this function will calculate the trend of a given array.
trend will calculate the avg of the first half of the array and then the avg of the second half, trend = avg2 - avg1.
for example:  [0,1,4,5,3,4,6,3] = 4 - 2.5 = 1.5
the function needs to be called:	array_trend(adr("array"),sizeof("array"));
because this function works with pointers its very time efficient and it needs no extra memory.

*)
stop := SHR(size,2)-1;
stop2 := SHR(stop,1);
FOR i := 0 TO stop2 DO x := x - pt^[i]; END_FOR;
IF EVEN(UINT_TO_INT(stop)) THEN
	FOR i := stop2 TO stop DO X := X + pt^[i]; END_FOR;
ELSE
	FOR i := stop2 + 1 TO stop DO X := X + pt^[i]; END_FOR;
END_IF;
ARRAY_TREND := x / (stop2 + 1);

(* revision history
hm	2 oct 2007	rev 1.0
	original version

hm	12 dec 2007	rev 1.1
	changed code for better performance

hm	16. mar. 2008	rev 1.2
	changed type of input size to uint

*)
END_FUNCTION

(* POU ASINH, ST *)
FUNCTION ASINH : REAL
VAR_INPUT
	X : REAL;
END_VAR
VAR
END_VAR


(*
version 1.2	16. mar 2008
programmer 	hugo
tested by		tobias

this function calculates the arcus sin hyperbolicus

*)
ASINH := LN(SQRT(X * X + 1)+X);

(* revision history
hm		12 jan 2007	rev 1.0
	original version

hm		2. dec 2007	rev 1.1
	changed code for better performance

hm		16.3. 2007		rev 1.2
	changed sequence of calculations to improve performance

*)
END_FUNCTION

(* POU ASTRO, ST *)
FUNCTION_BLOCK ASTRO
VAR_INPUT
	m : REAL;
	AE : REAL;
	PC : REAL;
	LJ : REAL;
END_VAR
VAR_OUTPUT
	Ym : REAL;
	YAE : REAL;
	YPC : REAL;
	YLJ : REAL;
END_VAR
VAR
END_VAR

(*
version 1.0	27 mar 2007
programmer 	hugo
tested by		oscat

this function converts different length units
any unused input can simply be left open.
different inputs connected at the same time will be added up.

*)
YAE :=	AE
		+ m / 149.597870E9
		+ PC * 206265
		+ LJ * 63240;
Ym := YAE * 149.597870E9;
YPC := YAE / 206265;
YLJ := YAE / 63240;


(*
Länge Meter m SI-Basiseinheit
Astronomische Einheit* AE 1 AE = 149,597 870 · E9 m
Parsec pc 1 pc = 206265 AE = 30,857 · E15 m
Lichtjahr Lj 1 Lj = 9,460 530 · E15 m = 63240 AE = 0,306 59 pc
Ångström Å 1 Å = E–l0 m
typograph. Punkt p 1 p = 0,376 065 mm • im Druckereigewerbe
inch** in 1 in = 2,54 · E–2 m = 25,4 mm***
foot ft 1 ft = 0,3048 m = 30,48 cm
yard yd 1 yd = 0,9144 m
mile mile 1 mile = 1609,344 m
Internat. Seemeile sm 1 sm = 1852 m
Fathom fm 1 fm = 1,829 m • in der Seeschifffahrt

*)
END_FUNCTION_BLOCK

(* POU ATAN2, ST *)
FUNCTION ATAN2 : REAL
VAR_INPUT
	Y : REAL;
	X : REAL;
END_VAR
VAR
END_VAR


(*
version 1.1	18. oct. 2008
programmer 	hugo
tested by	oscat

this function calculates the angle in a coordinate system in rad.

*)
IF X > 0 THEN
	ATAN2 := ATAN(Y/X);
ELSIF X < 0 THEN
	IF Y >=0 THEN
		ATAN2 := ATAN(Y/X) + MATH.PI;
	ELSE
		ATAN2 := ATAN(Y/X) - MATH.PI;
	END_IF;
ELSIF Y > 0 THEN
	ATAN2 := MATH.PI05;
ELSIF Y < 0 THEN
	ATAN2 := -MATH.PI05;
ELSE
	ATAN2 := 0;
END_IF;


(* revision history
hm	20.  apr. 2008	rev 1.0
	original version

hm	18. oct. 2008	rev 1.1
	changed to use math constants
*)
END_FUNCTION

(* POU ATANH, ST *)
FUNCTION ATANH : REAL
VAR_INPUT
	X : REAL;
END_VAR
VAR
END_VAR


(*
version 1.1	5. jan 2008
programmer 	hugo
tested by		tobias

this function calculates the arcus tangens hyperbolicus

*)
ATANH := LN((1+x)/(1-x)) * 0.5;


(* revision history
hm		12 jan 2007	rev 1.0
	original version

hm		5. jan 2008	rev 1.1
	improved code for better performance
*)
END_FUNCTION

(* POU B_TRIG, ST *)
FUNCTION_BLOCK B_TRIG
VAR_INPUT
	CLK : BOOL;
END_VAR
VAR_OUTPUT
	Q : BOOL;
END_VAR
VAR
	edge : BOOL;
END_VAR

(*
version 1.0	4. aug. 2006
programmer 	hugo
tested by		tobias

this block is similar to R_trig and F_trig but it generates a pulse on rising and falling edge.

*)
Q := clk XOR edge;
edge := CLK;


(* revision history
hm		4. aug. 2006	rev 1.0
	original version

*)
END_FUNCTION_BLOCK

(* POU BAR_GRAPH, ST *)
FUNCTION_BLOCK BAR_GRAPH
VAR_INPUT
	X : REAL;
	rst : BOOL;
END_VAR
VAR_INPUT CONSTANT
	trigger_Low : REAL;
	trigger_High : REAL;
	Alarm_low : BOOL;
	Alarm_high : BOOL;
	log_scale : BOOL;
END_VAR
VAR_OUTPUT
	LOW, Q1, Q2, Q3, Q4, Q5, Q6, HIGH : BOOL;
	Alarm : BOOL;
	Status : BYTE;
END_VAR
VAR
	init : BOOL;
	T1, T2, T3, T4, T5 : REAL;
END_VAR
VAR_TEMP
	temp : REAL;
END_VAR

(*
	version 1.2	6 jan 2008
	programmer 	hugo
	tested BY		hans

bar graph is a muti window comparator which displays an analog input signal on 8 digital outputs.
only one output is active a any given time depending on the value of the input signal.
the output can be of linear or logarithmic scale.

*)
IF NOT init THEN
	init := TRUE;
	IF log_scale THEN
		temp := EXP(LN(Trigger_high / Trigger_low) * 0.166666666666666666666);
		T1 := trigger_low * temp;
		T2 := T1 * temp;
		T3 := T2 * temp;
		T4 := T3 * temp;
		T5 := T4 * temp;
	ELSE
		temp := (trigger_high - trigger_low) * 0.142857142;
		T1 := trigger_low + temp;
		T2 := T1 + temp;
		T3 := T2 + temp;
		T4 := T3 + temp;
		T5 := T4 + temp;
	END_IF;
END_IF;

(* clear outputs before checking *)
Q1 := FALSE;
Q2 := FALSE;
Q3 := FALSE;
Q4 := FALSE;
Q5 := FALSE;
Q6 := FALSE;
status := 110;

(* low, high and alarm can only be cleared with rst depending on alarm_low and alarm_high *)
IF NOT alarm_low THEN low := FALSE; END_IF;
IF NOT alarm_high THEN high := FALSE; END_IF;
IF rst THEN
	alarm := FALSE;
	low := FALSE;
	high := FALSE;
END_IF;

(* check and set outputs *)
IF X < trigger_low THEN
	Low := TRUE;
	status := 111;
	IF alarm_low THEN
		alarm := TRUE;
		status := 1;
	END_IF;
ELSIF X < T1 THEN
	Q1 := TRUE;
ELSIF x < t2 THEN
	Q2 := TRUE;
ELSIF x < t3 THEN
	Q3 := TRUE;
ELSIF x < T4 THEN
	Q4 := TRUE;
ELSIF x < T5 THEN
	q5 := TRUE;
ELSIF x < trigger_high THEN
	q6 := TRUE;
ELSE
	high := TRUE;
	status := 112;
	IF alarm_high THEN
		alarm := TRUE;
		status := 2;
	END_IF;
END_IF;

(* revision history
hm	22. feb 2007	rev 1.0
	original version

hm	2. dec 2007		rev 1.1
	chaged code for better performance

hm	6. jan 2008		rev 1.2
	further performance improvement

*)
END_FUNCTION_BLOCK

(* POU BCDC_TO_INT, ST *)
FUNCTION BCDC_TO_INT : INT
VAR_INPUT
	IN : BYTE;
END_VAR
VAR
END_VAR

(*
version 1.1 30. jun. 2008
programmer 	hugo
tested by	oscat

this function converts a two digit bcd number into an integer.

*)
BCDC_TO_INT := (in AND 16#0F) + (SHR(in,4) * 10);

(* revision history
hm	13.12.2007	rev 1.0
	original version

hm	30.6.2008	rev 1.1
	changed name BCD_TO_INT to BCDC_TO_INT to avoid collision with util.lib

*)
END_FUNCTION

(* POU BETA, ST *)
FUNCTION BETA : REAL
VAR_INPUT
	X : REAL;
	Y : REAL;
END_VAR
VAR
END_VAR

(*
version 1.0	26. oct. 2008
programmer 	hugo
tested by		oscat

this function calculates the beta function for real number > 0.

*)
BETA := GAMMA(X) * GAMMA(Y) / GAMMA(x + y);


(* revision history
hm	26. oct. 2008	rev 1.0
	original version

*)
END_FUNCTION

(* POU GAMMA, ST *)
FUNCTION GAMMA : REAL
VAR_INPUT
	X : REAL;
END_VAR
VAR
END_VAR

(*
version 1.2	26. oct. 2008
programmer 	hugo
tested by	oscat

this function calculates the stirling function which is an approximation for the gamma function

*)
IF x > 0 THEN
	GAMMA := SQRT(math.PI2/X) * EXPT(math.E_INV * (x + 1 / (12 * x - 0.1 / X)),x);
END_IF;


(* the stirling formula is not very accurate for small values of X
IF X >=0 THEN GAMMA := SQRT(math.PI2 * X) * EXPT(X / math.E, X); END_IF;
*)





(* revision history
hm	10.12.2007	rev 1.0
	original version

hm	18. oct. 2008	rev 1.1
	using math constants

hm	26. oct. 2008	rev 1.2
	using new formula with better accuracy
*)
END_FUNCTION

(* POU BFT_TO_MS, ST *)
FUNCTION BFT_TO_MS : REAL
VAR_INPUT
	BFT : INT;
END_VAR
VAR
END_VAR

(*
version 1.0	12. jun 2008
programmer 	hugo
tested by	oscdat

this function converts wind speed from beaufort to m/s
*)
BFT_TO_MS := EXPT(BFT, 1.5) * 0.836;


(* revision history
hm	12. 6. 2008		rev 1.0
	original version

*)
END_FUNCTION

(* POU BIN_TO_BYTE, ST *)
FUNCTION BIN_TO_BYTE : BYTE
VAR_INPUT
	BIN : STRING(12);
END_VAR
VAR
	pt : POINTER TO BYTE;
	i: INT;
	X: BYTE;
	stop: INT;
END_VAR

(*
version 1.1	20. sep. 2008
programmer 	hugo
tested by	oscat

BINARY_TO_byte converts a binary string into a byte.

*)
pt := ADR(bin);
stop := LEN(bin);
FOR I := 1 TO stop DO
	(* read the first character and subtract 48 to get value in decimal 0 = 48 *)
	x := pt^;
	(* calculate the value of the digit *)
	IF X = 48 OR X = 49 THEN
		BIN_TO_BYTE := SHL(BIN_TO_BYTE,1) + X - 48;
	END_IF;
	pt := pt + 1;
END_FOR;



(* revision histroy
hm	18. jun. 2008	rev 1.0
	original release

hm	20. sep. 2008	rev 1.1
	changed length of input string from 20 to 12

*)	
END_FUNCTION

(* POU BIN_TO_DWORD, ST *)
FUNCTION BIN_TO_DWORD : DWORD
VAR_INPUT
	BIN : STRING(40);
END_VAR
VAR
	pt : POINTER TO BYTE;
	i: INT;
	X: BYTE;
	stop: INT;
END_VAR

(*
version 1.1	20. sep. 2008
programmer 	hugo
tested by	oscat

BINARY_TO_DWORD converts a binary string into a dword.

*)
pt := ADR(bin);
stop := LEN(bin);
FOR I := 1 TO stop DO
	(* read the first character and subtract 48 to get value in decimal 0 = 48 *)
	x := pt^;
	(* calculate the value of the digit *)
	IF X = 48 OR X = 49 THEN
		BIN_TO_DWORD := SHL(BIN_TO_DWORD,1) + X - 48;
	END_IF;
	pt := pt + 1;
END_FOR;



(* revision histroy
hm	18. jun. 2008	rev 1.0
	original release

hm	20. sep. 2008	rev 1.1
	changed length of input dtring from 20 to 40
*)	
END_FUNCTION

(* POU BINOM, ST *)
FUNCTION BINOM : DINT
VAR_INPUT
	N : INT;
	K : INT;
END_VAR

VAR
	i: INT;
END_VAR


(*
version 1.0	25. oct. 2008
programmer 	hugo
tested by		tobias

this function calculates the binomialkoefficient (N over k)

*)
IF 2 * K > n THEN
	k := n - k;
END_IF;
IF k > n THEN
	RETURN;
ELSIF k = 0 OR k = n THEN
	BINOM := 1;
ELSIF k = 1 THEN
	BINOM := n;
ELSE
	BINOM := n;
	n := n + 1;
	FOR i := 2 TO k DO
		BINOM := BINOM * (n - i) / i;
	END_FOR
END_IF;



(*
binomialkoeffizient(n, k)
1  wenn k = 0 return 1
2  wenn 2k > n
3      dann führe aus ergebnis \leftarrow binomialkoeffizient(n, n-k)
4  sonst führe aus ergebnis \leftarrow n
5          von i \leftarrow 2 bis k
6              führe aus ergebnis \leftarrow ergebnis \cdot (n + 1 - i)
7                        ergebnis \leftarrow ergebnis : i
8  return ergebnis
*)



(* revision history
hm	25. oct. 2008	rev 1.0
	original version


*)
END_FUNCTION

(* POU BIT_LOAD_B, ST *)
FUNCTION BIT_LOAD_B : BYTE
VAR_INPUT
	IN : BYTE;
	VAL : BOOL;
	POS : INT;
END_VAR
VAR CONSTANT
	dat : BYTE := 1;
END_VAR

(*
version 1.1	16. mar 2008
programmer 	hugo
tested by	tobias

this function loads a bit into a byte at position pos.
 *)
IF VAL THEN
	BIT_LOAD_B := in OR SHL(dat,pos);
ELSE
	BIT_LOAD_B := in AND (NOT SHL(dat,pos));
END_IF;


(* revision history
hm	29. feb 2008	rev 1.0
	original version

hm	16. mar 2008	rev 1.1
	change input bit to val for compatibility reasons
*)
END_FUNCTION

(* POU BIT_LOAD_B2, ST *)
FUNCTION BIT_LOAD_B2 : BYTE
VAR_INPUT
	I : BYTE;
	D : BOOL;
	P : INT;
	N : INT;
END_VAR


(*
version 1.0 18. oct. 2008
programmer 	hugo
tested by	tobias

this function loads N bits of D at pos P in Byte I

*)
IF D THEN
	BIT_LOAD_B2 := ROL(SHR(BYTE#255, 8 - N) OR ROR(i, P), P);
ELSE
	BIT_LOAD_B2 := ROL(SHL(BYTE#255, N) AND ROR(I, P), P);
END_IF;



(* revision history
hm	18. oct. 2008	rev 1.0
	original version


*)
END_FUNCTION

(* POU BIT_LOAD_DW, ST *)
FUNCTION BIT_LOAD_DW : DWORD
VAR_INPUT
	IN : DWORD;
	VAL : BOOL;
	POS : INT;
END_VAR
VAR CONSTANT
	dat : DWORD := 1;
END_VAR

(*
version 1.1	16. mar 2008
programmer 	hugo
tested by	tobias

this function loads a bit into a DWord at position pos.
 *)
IF val THEN
	BIT_LOAD_DW := in OR SHL(dat,pos);
ELSE
	BIT_LOAD_DW := in AND (NOT SHL(dat,pos));
END_IF;


(* revision history
hm	29. feb 2008	rev 1.0
	original version

hm	16. mar 2008	rev 1.1
	change input bit to val for compatibility reasons
*)
END_FUNCTION

(* POU BIT_LOAD_DW2, ST *)
FUNCTION BIT_LOAD_DW2 : DWORD
VAR_INPUT
	I : DWORD;
	D : BOOL;
	P : INT;
	N : INT;
END_VAR


(*
version 1.0 18. oct. 2008
programmer 	hugo
tested by	tobias

this function loads N bits of D at pos P in DWORD I

*)
IF D THEN
	BIT_LOAD_DW2 := ROL(SHR(DWORD#4294967295, 32 - N) OR ROR(i, P), P);
ELSE
	BIT_LOAD_DW2 := ROL(SHL(DWORD#4294967295, N) AND ROR(I, P), P);
END_IF;



(* revision history
hm	18. oct. 2008	rev 1.0
	original version


*)
END_FUNCTION

(* POU BIT_LOAD_W, ST *)
FUNCTION BIT_LOAD_W : WORD
VAR_INPUT
	IN : WORD;
	VAL : BOOL;
	POS : INT;
END_VAR
VAR CONSTANT
	dat : WORD := 1;
END_VAR

(*
version 1.1	16. mar 2008
programmer 	hugo
tested by	tobias

this function loads a bit into a Word at position pos.
 *)
IF val THEN
	BIT_LOAD_W := in OR SHL(dat,pos);
ELSE
	BIT_LOAD_W := in AND (NOT SHL(dat,pos));
END_IF;


(* revision history
hm	29. feb 2008	rev 1.0
	original version

hm	16. mar 2008	rev 1.1
	change input bit to val for compatibility reasons
*)
END_FUNCTION

(* POU BIT_LOAD_W2, ST *)
FUNCTION BIT_LOAD_W2 : WORD
VAR_INPUT
	I : WORD;
	D : BOOL;
	P : INT;
	N : INT;
END_VAR


(*
version 1.0 18. oct. 2008
programmer 	hugo
tested by	tobias

this function loads N bits of D at pos P in WORD I

*)
IF D THEN
	BIT_LOAD_W2 := ROL(SHR(WORD#65535, 16 - N) OR ROR(i, P), P);
ELSE
	BIT_LOAD_W2 := ROL(SHL(WORD#65535, N) AND ROR(I, P), P);
END_IF;



(* revision history
hm	18. oct. 2008	rev 1.0
	original version


*)
END_FUNCTION

(* POU BIT_OF_DWORD, ST *)
FUNCTION BIT_OF_DWORD : BOOL
VAR_INPUT
	in : DWORD;
	N : INT;
END_VAR
VAR
END_VAR

(*
version 1.2	6. jun. 2008
programmer 	hugo
tested by	tobias

this function extracts a single bit from the nth position from right (right is lowest bit)
the lowest Bit (Bit0 from in) is selected with N=0.
 *)
BIT_OF_DWORD := (SHR(in,N) AND 16#00000001) > 0;


(* old code used before rev 1.1
temp := SHR(in,n);
Bit_of_Dword := temp.0;
*)


(* revision history
hm	4. aug. 2006	rev 1.0
	original version

hm	29. feb 2008	rev 1.1
	improved performance

hm	6. jun. 2008	rev 1.2
	changes type of input N from byte to int
*)
END_FUNCTION

(* POU BIT_TOGGLE_B, ST *)
FUNCTION BIT_TOGGLE_B : BYTE
VAR_INPUT
	IN : BYTE;
	POS : INT;
END_VAR


(*
version 1.0 18. oct. 2008
programmer 	hugo
tested by	tobias

this function toggles a bit of a BYTE at position pos.

*)
BIT_TOGGLE_B := SHL(BYTE#1, POS) XOR IN;




(* revision history
hm	18. oct. 2008	rev 1.0
	original version


*)
END_FUNCTION

(* POU BIT_TOGGLE_DW, ST *)
FUNCTION BIT_TOGGLE_DW : DWORD
VAR_INPUT
	IN : DWORD;
	POS : INT;
END_VAR


(*
version 1.0 18. oct. 2008
programmer 	hugo
tested by	tobias

this function toggles a bit of a WORD at position pos.

*)
BIT_TOGGLE_DW := SHL(DWORD#1, POS) XOR IN;



(* revision history
hm	18. oct. 2008	rev 1.0
	original version


*)
END_FUNCTION

(* POU BIT_TOGGLE_W, ST *)
FUNCTION BIT_TOGGLE_W : WORD
VAR_INPUT
	IN : WORD;
	POS : INT;
END_VAR


(*
version 1.0 18. oct. 2008
programmer 	hugo
tested by	tobias

this function toggles a bit of a WORD at position pos.

*)
BIT_TOGGLE_W := SHL(WORD#1, POS) XOR IN;



(* revision history
hm	18. oct. 2008	rev 1.0
	original version


*)
END_FUNCTION

(* POU BLIND_ACTUATOR, ST *)
 FUNCTION_BLOCK BLIND_ACTUATOR
VAR_INPUT
	UP, DN : BOOL;
	S_IN : BYTE;
	T_UD : TIME := T#10s;
	T_ANGLE : TIME := T#3s;
END_VAR
VAR_INPUT CONSTANT
	T_LOCKOUT : TIME := t#100ms;
END_VAR
VAR_OUTPUT
	POS, ANG : BYTE;
	QU, QD : BOOL;
	STATUS : BYTE;
END_VAR
VAR
	position, angle : RMP_B;
	lock : INTERLOCK;
END_VAR

(*
version 1.2	18. oct. 2008
programmer 	hugo
tested by	oscat

blind actuator drives the up and down motor of a blind. T_lockout specifies the time between up or dn becomes active. 
To change direction there must be a minimum wait time to allow the motors to come to rest first.
the up and down outputs QU and QD are controlled by the inputs UP and DN.
the outputs pos and ang simulate the position of the blind pos = 0 means blind is down and pos = 255 = blind is up.
the angle 0 means vertical posisition of the slates and 255 means horizontal position of the slates.


*)
(* make sure only one motor is active at a given time *)
lock(i1 := UP, I2 := DN, TL := T_lockout);

(* ramp up or down to simulate the angle position of the blind slats *)
angle(e := lock.Q1 OR lock.Q2, UP := lock.Q1, PT := T_Angle);
position(e := lock.Q1 AND angle.high OR lock.Q2 AND angle.low, up := lock.Q1, PT := T_UD);

(* set the outputs *)
pos := position.Out;
ang := angle.Out;
QU := lock.Q1;
QD := lock.Q2;

(* set the status output *)
IF UP AND DN THEN
	IF s_in < 10 AND S_in > 1 THEN status := s_in; ELSE status := 1; END_IF;			(* error up and down together are not allowed *)
ELSIF S_IN > 0 THEN
	status := S_IN;
ELSIF UP THEN
	status := 101;
ELSIF DN THEN
	status := 102;
ELSE
	status := 0;
END_IF;


(* revision history
hm	29. sep 2007	rev 1.0
	original release

hm	6. oct 2007		rev 1.1
	rearanged outputs

hm	18. oct. 2008	rev 1.2
	changed calls for rmp_B because of change in RMP_B
*)
END_FUNCTION_BLOCK

(* POU RMP_B, ST *)
FUNCTION_BLOCK RMP_B
VAR_INPUT
	SET : BOOL;
	PT : TIME;
	E : BOOL := TRUE;
	UP : BOOL := TRUE;
	RST : BOOL;
END_VAR
VAR_OUTPUT
	OUT : BYTE;
	BUSY: BOOL;
	HIGH : BOOL;
	LOW : BOOL;
END_VAR
VAR
	rmp : _RMP_B;
END_VAR


(*
version 2.0	23. oct. 2008
programmer 	oscat
tested BY	oscat

this ramp generator generates a byte wide ramp with 255 steps
the generator has an asynchronous set and reset
the ramp is controlled by PT which is the total ramp time for a full sweep from 0..255
an UD input controlls the direction Up or Down and the E input enables the ramp generation
a busy output indicates that the ramp is running, busy false means output is stable.
the outputs low and high will be true when the output has reached its max or min value.

*)
(* generate ramp *)
rmp(dir := UP, E := E, TR := PT, rmp := out);

(* set or reset operation *)
IF RST THEN
	out := 0;
ELSIF SET THEN
	out := 255;
END_IF;

(* checks for outputs stable and reset or set busy flag *)
low := out = 0;
high := out = 255;
busy := NOT (low OR high) AND E;


(* revision history

hm 5.10.2006	rev 1.1
	added busy output
hm 17.1.2007	rev 1.2
	renamed input ud to up for better usability
	deleted unused variable step

hm	17.9.2007		rev 1.3
	replaced time() with t_plc_ms() for compatibility reasons

hm	28. sep 2007	rev 1.4
	added outputs on and off
	busy is now disabled while en is false
	new coding for higher accuracy and performance

hm	5. oct 2007	rev 1.5
	added statements to allow for PT to be t#0s output jumps to max or min immediately

hm	25. dec 2007	rev 1.6
	improved code for better performance

hm	16. oct. 2008	rev 1.7
	improved code for better performance

hm	18. oct. 2008	rev 1.8
	added type conversion to avoid warnings
	changed input en to e for compatibility reasons

hm	23. oct. 2008	REV 	2.0
	new code using _RMP_B

*)
END_FUNCTION_BLOCK

(* POU INTERLOCK, ST *)
FUNCTION_BLOCK INTERLOCK
VAR_INPUT
	I1, I2 : BOOL;
	TL : TIME;
END_VAR
VAR_OUTPUT
	Q1, Q2 : BOOL;
END_VAR
VAR
	T1, T2 : TOF;
END_VAR

(*
version 1.0	28 sep 2007
programmer 	hugo
tested by		tobias

INTERLOCK has two inputs I1 and I2 which drive the corresponding outputs Q1 and Q2.
the inputs signals lock each other out and therfore I1 can only drive Q1 when I2 is Low and vice versa.
The input TL specifies a dead time between two outputs can become active.
an output can only become active when the other output was not active for the time TL.

*)
(* the input signal have a run delay to lockout the other input *)
T1(IN := I1, PT := TL);
T2(IN := I2, PT := TL);

Q1 := I1 AND NOT t2.Q;
Q2 := I2 AND NOT t1.Q;


(* revision history

hm	28 sep 2007		rev 1.0
	original version

*)
END_FUNCTION_BLOCK

(* POU BLIND_CONTROL, ST *)
FUNCTION_BLOCK BLIND_CONTROL
VAR_INPUT
	UP, DN : BOOL;
	S_IN : BYTE;
	PI : BYTE;
	AI : BYTE;
	T_UD, T_ANGLE : TIME;
END_VAR
VAR_INPUT CONSTANT
	SENS : BYTE := 5;
	T_LOCKOUT: TIME := T#100ms;
END_VAR
VAR_OUTPUT
	POS, ANG : BYTE;
	MU, MD : BOOL;
	STATUS : BYTE;
END_VAR
VAR
	act : BLIND_ACTUATOR;
	delta : BYTE;
END_VAR

(*
version 1.3	30. oct 2007
programmer 	hugo
tested by		tobias


*)
IF UP AND DN THEN
	(* automatic modus detected *)
	(* first find correct position *)
	IF BYTE_TO_INT(act.pos) < BYTE_TO_INT(pi) - delta THEN
		act.UP := TRUE;
		act.DN := FALSE;
		delta := 0;
		act.S_IN := 121;
	ELSIF BYTE_TO_INT(act.pos) > BYTE_TO_INT(pi) + delta THEN
		act.UP := FALSE;
		act.DN := TRUE;
		delta := 0;
		act.S_IN := 122;
	(* regulate angle *)
	ELSIF BYTE_TO_INT(act.ang) < BYTE_TO_INT(ai) - delta AND T_angle > T#100ms THEN
		act.UP := TRUE;
		act.DN := FALSE;
		delta := 0;
		act.S_IN := 123;
	ELSIF BYTE_TO_INT(act.ang) > BYTE_TO_INT(ai) + delta AND T_angle > T#100ms THEN
		act.UP := FALSE;
		act.DN := TRUE;
		delta := 0;
		act.S_IN := 124;
	(* correct position reached *)
	ELSE
		act.UP := FALSE;
		act.DN := FALSE;
		delta := sens;
		act.S_IN := 0;
	END_IF;
ELSE
	act.UP := UP;
	act.DN := DN;
END_IF;

(* hand over status *)
IF s_in > 0 THEN act.S_IN := S_IN; END_IF;

(* blind control calls blind_actuator *)
act(T_UD:=T_UD, T_ANGLE:=T_ANGLE, T_lockout := T_Lockout);
pos := act.pos;
ang := act.ang;
MU := act.QU;
md := act.QD;
status := act.status;

(* revision history
hm	29. sep 2007	rev 1.0
	original release

hm	6. oct 2007		rev 1.1
	rearranged outputs
	integrated blind_actuator into blind_control

hm	16. oct 2007	rev 1.2
	ignore angle when t_angle = 0

hm 29. oct 2007	rev 1.3
	added lockout configuration time for motor direction change
	sens has a setup value of 5
*)
END_FUNCTION_BLOCK

(* POU BLIND_INPUT, ST *)
FUNCTION_BLOCK BLIND_INPUT
VAR_INPUT
	POS, ANG : BYTE;
	S1, S2 : BOOL;
	IN : BOOL;
	PI, AI : BYTE;
END_VAR
VAR_INPUT CONSTANT
	SINGLE_SWITCH : BOOL;
	CLICK_EN : BOOL := TRUE;
	CLICK_TIME : TIME := T#500ms;
	MAX_RUNTIME : TIME := T#60s;
	MANUAL_TIMEOUT: TIME := T#1h;
	DEBOUNCE_TIME : TIME := T#20ms;
	DBL_CLK1 : BOOL := FALSE;
	DBL_POS1 : BYTE;
	DBL_ANG1 : BYTE;
	DBL_CLK2 : BOOL := FALSE;
	DBL_POS2 : BYTE := 255;
	DBL_ANG2 : BYTE := 255;
	D1_TOGGLE : BOOL := TRUE;
	D2_TOGGLE : BOOL := TRUE;
END_VAR
VAR_OUTPUT
	QU, QD : BOOL;
	STATUS : BYTE;
	PO, AO : BYTE;
	D1, D2 : BOOL;
END_VAR
VAR
	s1e, s2e : TOF;
	s1d, s2d : CLICK_MODE;
	dir : BOOL;
	tx, last : TIME;
END_VAR

(*
version 1.5	22. jan. 2009
programmer 	hugo
tested by		oscat


*)
(* read system timer *)
tx := DWORD_TO_TIME(T_PLC_MS());

(* inputs S1 and S2 are debounced and then decoded for multiple clicks *)
s1e(in := S1, pt := DEBOUNCE_TIME);
s2e(in := S2, pt := DEBOUNCE_TIME);
s1d(in := (s1e.Q AND NOT SINGLE_SWITCH) OR (s1e.Q AND SINGLE_SWITCH AND dir), t_long := CLICK_TIME);
s2d(in := (s2e.Q AND NOT SINGLE_SWITCH) OR (s1e.Q AND SINGLE_SWITCH AND NOT dir), t_long := CLICK_TIME);

(* if d1 and d2 are not toggle clear them to make sure they are only active for oine cycle *)
IF NOT d1_toggle THEN d1 := FALSE; END_IF;
IF NOT d2_toggle THEN d2 := FALSE; END_IF;

(* decode actions *)
IF s1d.tp_LONG THEN
	status := 132;
ELSIF s2d.tp_LONG THEN
	status := 133;
ELSIF  s1d.SINGLE THEN
	IF click_en THEN
		(* if running then we stop otherwise start new direction *)
		IF QU XOR QD THEN
			status := 131;
		ELSE
			status := 134;
			last := tx;
			dir := NOT dir;
		END_IF;
	END_IF;
ELSIF  s2d.SINGLE THEN
	IF click_en THEN
		(* if running then we stop otherwise start new direction *)
		IF QU XOR QD THEN
			status := 131;
		ELSE
			status := 135;
			last := tx;
			dir := NOT dir;
		END_IF;
	END_IF;
ELSIF in THEN
	status := 136;
	last := tx;
ELSIF s1d.DOUBLE THEN
	IF dbl_clk1 THEN
		(* a position need to be set for a double click on S1 *)
		status := 137;
		last := tx;
	ELSE
		(* toggle the output when dbl_clk1 is not active *)
		D1 := NOT D1;
	END_IF;
ELSIF s2d.DOUBLE THEN
	IF dbl_clk2 THEN
		(* a position need to be set for a double click on S2 *)
		status := 138;
		last := tx;
	ELSE
		(* toggle the output when dbl_clk2 is not active *)
		(* in single switch mode we need to toggle d1 instead of d2 *)
		IF single_switch THEN D1 := NOT D1; ELSE D2 := NOT D2; END_IF;
	END_IF;
END_IF;


(* state machine *)
CASE status OF
	0:	(* automatic standby operation *)
			QU := QD := TRUE;
			PO := POS; AO := ANG;
	131:	(* manual operation standby *)
			QU := QD := FALSE;
			(* manual mode will be ended when timeout is reached *)
			IF tx - last >= manual_timeout THEN status := 0; END_IF;
	132:	(* manual operation up *)
			QU := TRUE; QD := FALSE;
			PO := POS; AO := ANG;
			last := tx;
			IF NOT s1d.LONG THEN status := 131; dir := NOT dir; END_IF;
	133:	(* manual operation down *)
			QU := FALSE; QD := TRUE;
			PO := POS; AO := ANG;
			last := tx;
			IF NOT s2d.LONG THEN	status := 131; dir := NOT dir; END_IF;
	134:	(* manual operation single click up *)
			QU := TRUE; QD := FALSE;
			PO := POS; AO := ANG;
			IF tx - last >= max_runtime THEN status := 131; END_IF;
	135:	(* manual operation single click dn *)
			QU := FALSE; QD := TRUE;
			PO := POS; AO := ANG;
			IF tx - last >= max_runtime THEN status := 131;	END_IF;
	136:	(* forced input in = true *)
			QU := QD := TRUE;
			PO := PI; AO := AI;
			IF tx-last >= max_runtime THEN status := 0; END_IF;
	137:	(* double click1 position *)
			QU := QD := TRUE;
			PO := DBL_POS1;
			AO := DBL_ANG1;
			IF tx - last >= max_runtime THEN status := 131; END_IF;
	138:	(* double click2 position *)
			QU := QD := TRUE;
			PO := DBL_POS2;
			AO := DBL_ANG2;
			IF tx - last >= max_runtime THEN status := 131; END_IF;
END_CASE




(* revision history
hm	29. sep 2007	rev 1.0
	original release

hm	6. oct 2007		rev 1.1
	renamed ps and as to po and ao

hm	30. dec 2007	rev 1.2
	added click_timeout variable and function

hm	16. jul. 2008	rev 1.3
	rewirtten code to allow for more functionality
	added single click mode with single_switch.
	added Debounce for inputs S1 and S2
	added double_click functionality

hm	26. sep. 2008	rev 1.4
	corrected an error while POS and ANG was transferred to outputs PO and AO during automatic modes

hm	22. jan 2009	rev 1.5
	added pulse mode for double click outputs
	added automatic mode for IN
*)
END_FUNCTION_BLOCK

(* POU CLICK_MODE, ST *)
FUNCTION_BLOCK CLICK_MODE
VAR_INPUT
	IN : BOOL;
END_VAR
VAR_OUTPUT
	SINGLE : BOOL;
	DOUBLE : BOOL;
	LONG : BOOL;
	TP_LONG : BOOL;
END_VAR
VAR_INPUT CONSTANT
	T_LONG : TIME := t#500ms;
END_VAR
VAR
	Timer : TP;
	cnt : INT;
	last : BOOL;
END_VAR


(*
version 1.0	13. nov. 2008
programmer 	oscat
tested by	hugo

click_mode decodes an input for single, double or long click and sets the corresponding output single, doulbe or long.
the input configures itself to be high or low active depending on which state the input stays longer than t_reconfig.

*)
(* when input goes high start the timer to decode pulses *)
timer(in := IN, PT := T_LONG);
single := double := FALSE;

IF timer.Q THEN
	(* decode pulses while the timer is active *)
	IF NOT in AND last THEN	cnt := cnt + 1; END_IF;
ELSE
	CASE cnt OF
		1 : single := TRUE;
		2 : double := TRUE;
	END_CASE;
	cnt := 0;
END_IF;
last := in;
TP_LONG := NOT timer.Q AND (NOT LONG) AND IN;
LONG := NOT timer.Q AND in;




(* revision history

hm	13. nov. 2008	rev 1.0
	original release

*)
END_FUNCTION_BLOCK

(* POU BLIND_NIGHT, ST *)
FUNCTION_BLOCK BLIND_NIGHT
VAR_INPUT
	UP, DN : BOOL;
	S_IN : BYTE;
	PI, AI : BYTE;
	E_NIGHT : BOOL := TRUE;
	E_DAY	: BOOL := TRUE;
	DTIN : DT;
	SUNRISE, SUNSET : TOD;
END_VAR
VAR_INPUT CONSTANT
	sunrise_offset : TIME;
	sunset_offset : TIME;
	night_position : BYTE;
	night_angle : BYTE;
END_VAR
VAR_OUTPUT
	QU, QD : BOOL;
	STATUS : BYTE;
	PO, AO : BYTE;
END_VAR
VAR
	night : BOOL;
	last_night, last_day : DATE;
END_VAR

(*
version 1.2	6 oct 2007
programmer 	hugo
tested by		tobias


*)
IF NOT (up AND dn) AND night THEN
	(* manual operation at night will cancel operation for one night *)
	night := FALSE;
ELSIF (DT_TO_TOD(dtin) > sunset + sunset_offset) AND (last_night < DT_TO_DATE(dtin)) AND NOT night AND e_night THEN
	(* enable night *)
	night := TRUE;
	last_night := DT_TO_DATE(dtin);
ELSIF (DT_TO_TOD(dtin) > sunrise + sunrise_offset) AND (last_day < DT_TO_DATE(dtin)) AND night AND e_day AND (last_night < DT_TO_DATE(dtin)) THEN
	(* disable night *)
	night := FALSE;
	last_day := DT_TO_DATE(dtin);
END_IF;

(* shade at night only in auto mode and enable = true *)
IF UP AND DN AND night THEN
	status := 141;
	po := night_position;
	ao := night_angle;
ELSE
	QU := UP;
	QD := DN;
	po := pi;
	ao := ai;
	status := s_in;
END_IF;


(* revision history
hm	29. sep 2007	rev 1.0
	original version

hm	5. oct 2007		rev 1.1
	added enable input

hm	6. oct 2007		rev 1.2
	added pos and angle inputs and outputs
	night position and angle can now be configured
	any manual operation at night will cancel night operation

*)
END_FUNCTION_BLOCK

(* POU BLIND_SCENE, ST *)
FUNCTION_BLOCK BLIND_SCENE
VAR_INPUT
	UP, DN : BOOL;
	S_IN : BYTE;
	PI, AI : BYTE;
	ENABLE : BOOL;
	SWRITE : BOOL;
	SCENE : BYTE;
END_VAR
VAR_INPUT CONSTANT
END_VAR
VAR_OUTPUT
	QU, QD : BOOL;
	STATUS : BYTE;
	PO, AO : BYTE;
END_VAR
VAR RETAIN
	sx : ARRAY[0..15,0..2] OF BYTE;
END_VAR
VAR_TEMP
	x : BYTE;
END_VAR

(*
version 1.1	29. jan 2008
programmer 	hugo
tested by		tobias


*)
(* delete all bits except the lower 4 of scene *)
x := scene AND 16#0F;

IF enable AND sx[x,2] > 0 AND UP AND DN THEN
	po := sx[x,0];
	ao := sx[x,1];
	status := 160 + x;  (* Status number is 160 to 175 for the 16 scenes *)
	QU := TRUE;
	QD := TRUE;
ELSE
	QU := UP;
	QD := DN;
	status := S_IN;
	po := pi;
	ao := ai;
END_IF;

(* write scene if necessary *)
IF swrite THEN
	status := 176;		(* write scene *)
	sx[x,0] := pi;
	sx[x,1] := ai;
	IF enable THEN sx[x,2] := 1; ELSE sx[x,2] := 0; END_IF; (* if sx[x,2] = 0 the scene is disabled *)
END_IF;


(* revision history
hm	24. oct 2007	rev 1.0
	original release

hm		29.1.2008	rev 1.1
	replaced shr/shl with and for better performance
*)
END_FUNCTION_BLOCK

(* POU BLIND_SECURITY, ST *)
FUNCTION_BLOCK BLIND_SECURITY
VAR_INPUT
	UP, DN : BOOL;
	S_IN : BYTE;
	PI, AI : BYTE;
	FIRE : BOOL;
	WIND : BOOL;
	ALARM : BOOL;
	DOOR : BOOL;
	RAIN : BOOL;
END_VAR
VAR_INPUT CONSTANT
	Alarm_UP : BOOL := TRUE;
	WIND_UP :BOOL := TRUE;
	RAIN_UP : BOOL := FALSE;
END_VAR
VAR_OUTPUT
	QU, QD : BOOL;
	STATUS : BYTE;
	PO, AO : BYTE;
END_VAR
VAR
END_VAR

(*
version 1.2	12. feb 2008
programmer 	hugo
tested by		tobias


*)
IF Fire THEN
	QU := TRUE;
	QD := FALSE;
	status := 111;
ELSIF Wind THEN
	QU := Wind_up;
	QD := NOT wind_up;
	status := 112;
ELSIF alarm THEN
	QU := Alarm_up;
	QD := NOT Alarm_up;
	status := 113;
ELSIF Door THEN
	QU := TRUE;
	QD := FALSE;
	status := 114;
ELSIF Rain AND NOT (up XOR dn) THEN
	QU := rain_up;
	QD := NOT rain_up;
	status := 115;
ELSE
	QU := UP;
	QD := DN;
	status := S_IN;
	po := pi;
	ao := ai;
END_IF;


(* revision history
hm	29. sep 2007	rev 1.0
	original release

hm	6. oct 2007		rev 1.1
	added pos and angle inputs and outputs
	manual will override rain position
	alarm position can now be configured

hm		12. feb. 2008	rev 1.2
	added config variables rain_up and wind_up
	position for rain and wind is now configurable
*)
END_FUNCTION_BLOCK

(* POU BLIND_SHADE, ST *)
FUNCTION_BLOCK BLIND_SHADE
VAR_INPUT
	UP, DN : BOOL;
	S_IN : BYTE;
	PI, AI : BYTE;
	ENABLE : BOOL;
	SUN : BOOL;
END_VAR
VAR_IN_OUT
	CX : calendar;
END_VAR
VAR_INPUT CONSTANT
	sunrise_offset : TIME := T#1h;
	sunset_preset : TIME := T#1h;
	direction : REAL := 180;
	angle_offset : REAL := 80;
	slat_width : REAL := 80;
	Slat_spacing : REAL := 60;
	Shade_delay : TIME := T#60s;
	Shade_pos : BYTE;
END_VAR
VAR_OUTPUT
	QU, QD : BOOL;
	STATUS : BYTE;
	PO, AO : BYTE;
END_VAR
VAR
	angle: REAL;
	sun_delay : TOF;
END_VAR

(*
version 1.3	8. feb 2009
programmer 	hugo
tested by		tobias


*)
(* the input sun is sent through tof which will delay the shade for the time shade_delay *)
sun_delay(IN := sun, PT := shade_delay);

IF UP AND DN AND enable AND sun_delay.Q AND cx.SUN_HOR > direction - angle_offset AND cx.SUN_HOR < direction + angle_offset AND
	DT_TO_TOD(cx.UTC) > cx.SUN_RISE + sunrise_offset AND DT_TO_TOD(cx.UTC) < cx.SUN_SET - sunset_preset THEN
	status := 151;
	QU := UP;
	QD := DN;
	(* position is predefined *)
	po := shade_pos;
	(* shading is active now calculate the slat angle *)
	(* calculate the max angle for the blind *)
	angle := DEG(ATAN(slat_spacing / slat_width));
	(* check if sun angle is between 0 and max angle *)
	IF cx.SUN_VER > 0 AND cx.SUN_VER < angle THEN
		angle := cx.SUN_VER + DEG(ACOS(COS(RAD(cx.SUN_VER))*slat_spacing / Slat_width));
		ao := INT_TO_BYTE(LIMIT(0,TRUNC(angle * 255 / 90), 255));
	ELSE
		ao := 255;
	END_IF;
ELSE
	QU := UP;
	QD := DN;
	po := pi;
	ao := ai;
	status := S_IN;
END_IF;

(* revision history
hm	15 oct. 2007	rev 1.0
	original version

hm	19. oct 2007	rev 1.1
	manual mode was not detected because outputs were checked and not inputs UP and DN

hm	24. nov 2007	rev 1.2
	added shade_delay to avoid constant up and down if sun is out parcially

hm	8. feb 2009	rev 1.3
	added shading position shade_pos to be configured
	changed inputs to utilize calendar data structure

*)
END_FUNCTION_BLOCK

(* POU DEG, ST *)
FUNCTION DEG : REAL
VAR_INPUT
	rad : REAL;
END_VAR
VAR
END_VAR
VAR
END_VAR

(*
version 1.1	16 oct 2007
programmer 	hugo
tested by		tobias

this function converts degrees into Radiant
execution time on wago 750 - 841 =  10  us
*)
deg := modR(57.29577951308232 * Rad, 360);

(* revision history
hm	4. aug 2006		rev 1.0
	original version

hm 	16. oct 2007	rev 1.1
	added modr statement which prohibits deg to become bigger than 360

*)
END_FUNCTION

(* POU RAD, ST *)
FUNCTION RAD : REAL
VAR_INPUT
	deg : REAL;
END_VAR
VAR
END_VAR

(*
version 1.2	18. oct. 2008
programmer 	hugo
tested by	tobias

this function converts Radiant to degrees

*)
RAD := MODR(0.0174532925199433 * DEG, math.PI2);

(* revision history
hm	4. aug 2006		rev 1.0
	original version

hm 	16. oct 2007	rev 1.1
	added modr statement which prohibits rad to become bigger than 2PI

hm	18. oct 2008	rev 1.2
	using math constants

*)
END_FUNCTION

(* POU MODR, ST *)
FUNCTION MODR : REAL
VAR_INPUT
	IN : REAL;
	DIVI : REAL;
END_VAR

VAR
END_VAR

(*
version 1.4	31. oct. 2008
programmer 	hugo
tested by	tobias

this is a modulo funtion for real numbers
modr(5.5,2.5) = 0.5

*)
IF divi = 0 THEN
	MODR := 0;
ELSE
	MODR := in - DINT_TO_REAL(FLOOR2(in / divi)) * divi;
END_IF;

(* revision history

hm	4. aug.2006		rev 1.0

hm	28. jan.2007	rev 1.1
	modr(x,0) will deliver the result 0

hm	21. mar 2008	rev 1.2
	use D_trunc for compatibility reasons

hm	4. apr. 2008	rev 1.3
	added type conversion to avoid warnings under codesys 3.0

hm	31. oct. 2008	rev 1.4
	changed algorithm to the more common version using floor instead of TRUNC
*)
END_FUNCTION

(* POU FLOOR2, ST *)
FUNCTION FLOOR2 : DINT
VAR_INPUT
	X : REAL;
END_VAR
VAR
END_VAR


(*
version 1.1	4. apr. 2008
programmer 	hugo
tested by		tobias

This is a rounding function which returns the biggest possible integer which is less or equal to X.
floor2(3.14) = 3
floor2(-3.14) = -4

*)
FLOOR2 := REAL_TO_DINT(X);
IF DINT_TO_REAL(FLOOR2) > X THEN
	FLOOR2 := FLOOR2 - 1;
END_IF;

(* revision history
hm	21. mar. 2008	rev 1.0
	originlal version

hm	4. apr. 2008	rev 1.1
	added type conversion to avoid warnings under codesys 3.0
*)
END_FUNCTION

(* POU BOILER, ST *)
FUNCTION_BLOCK BOILER
VAR_INPUT
	T_upper : REAL;
	T_lower : REAL;
	Pressure : BOOL := TRUE;
	enable : BOOL := TRUE;
	Req_1 : BOOL;
	Req_2 : BOOL;
	Boost : BOOL;
END_VAR
VAR_INPUT CONSTANT
	t_upper_min : REAL := 50;
	t_upper_max : REAL := 60;
	T_lower_enable : BOOL;
	T_lower_max : REAL := 60;
	T_request_1 : REAL := 70;
	T_request_2 : REAL := 50;
	T_request_hys : REAL := 5;
	T_protect_high : REAL := 80;
	T_protect_low : REAL := 10;
END_VAR
VAR_OUTPUT
	Heat : BOOL;
	error : BOOL;
	status : BYTE;
END_VAR
VAR
	edge: BOOL;
	boost_mode: BOOL;
	flag_0 : BOOL;
	flag_1: BOOL;
	flag_2: BOOL;
END_VAR

(*
version 1.1	16. oct. 2008
programmer 	hugo
tested by	oscat


this function block controls a hot water boiler. The Boiler can be equipped with two temperature sensors on top and bottom of the tank, T_LOWER_ENABLE must be set to True in this case.
alternatively can BOILER be configured for one (TOP) temperature sensor only (T_LOWER_ENABLE set to False).
A Pressure sensor is used to detect fresh water pressure and disable all heating if there is no water pressure. This input is dset to True by default, so if it is not used it can simply be left open.
A enable input enables the hot water heating while it is set to True. alternatively can a Ture on Req_1 or Req_2 start the heating to predefined temperatures during setup.
A low to high edge on the boost input will start heating imediately until T_upper_max is reached, it can be used to generate extra hot water when needed.

*)
(* read sensors and check for valid data *)
IF t_upper > t_protect_high THEN
	status := 1;
	heat := FALSE;
	error := TRUE;
ELSIF t_upper < t_protect_low THEN
	status := 2;
	heat := error := TRUE;
ELSIF t_lower > T_protect_high AND t_lower_enable THEN
	status := 3;
	heat := FALSE;
	error := TRUE;
ELSIF t_lower < t_protect_low AND t_lower_enable THEN
	status := 4;
	heat := error := TRUE;
ELSIF NOT pressure THEN
	status := 5;
	heat := FALSE;
	error := TRUE;
ELSIF req_1 OR req_2 OR enable OR boost THEN
	error := FALSE;

	(* determine if heat needs to be turned on *)
	IF boost AND NOT edge AND t_upper < t_upper_max THEN
		status := 101;
		heat := TRUE;
		boost_mode := TRUE;
	ELSIF enable AND t_upper < T_upper_min THEN
		status := 102;
		heat := TRUE;
	ELSIF req_1 AND t_upper < T_request_1 THEN
		status := 103;
		heat := TRUE;
	ELSIF req_2 AND t_upper < t_request_2 THEN
		status := 104;
		heat := TRUE;
	END_IF;

	(* determine the shut off temperature *)
	IF heat THEN
		IF (enable OR boost_mode) THEN
			flag_0 := TRUE;
			IF T_lower_enable AND T_lower > T_lower_max THEN
				flag_0 := boost_mode := FALSE;
			ELSIF NOT T_lower_enable AND T_upper > T_upper_max THEN
				flag_0 := boost_mode := FALSE;
			END_IF;
		ELSE
			flag_0 := FALSE;
		END_IF;
		flag_1 := (req_1 AND T_upper > T_request_1 + T_request_hys) AND req_1;
		flag_2 := (req_2 AND T_upper > T_request_2 + T_request_hys) AND req_2;

		(* shut off heat if no longer needed *)
		heat := flag_0 OR flag_1 OR flag_2;
		IF heat = FALSE THEN status := 100; END_IF;
	END_IF;
ELSE
	status := 100;
	heat := error := FALSE;
END_IF;
edge := boost;


(* revision history
hm	27. feb. 2007	rev 1.0
	original version

hm	16. oct. 2008	rev 1.1
	improved performance


*)
END_FUNCTION_BLOCK

(* POU PRESSURE, ST *)
FUNCTION_BLOCK PRESSURE
VAR_INPUT
	mws : REAL;
	torr : REAL;
	att : REAL;
	atm : REAL;
	pa : REAL;
	bar : REAL;
END_VAR
VAR_OUTPUT
	Ymws : REAL;
	Ytorr : REAL;
	Yatt : REAL;
	Yatm : REAL;
	Ypa : REAL;
	Ybar : REAL;
END_VAR
VAR
END_VAR

(*
version 1.0	27 mar 2007
programmer 	hugo
tested by		oscat

this function converts different pressure units
any unused input can simply be left open.
different inputs connected at the same time will be added up.
*)
Ybar := bar +
		pa / 100000 +
		0.980665 * att +
		1.01325 * atm +
		0.001333224 * torr +
		0.0980665 * mws;
Ymws := ybar / 0.0980665;
Ytorr := ybar / 0.001333224;
Yatt := ybar / 0.980665;
yatm := ybar / 1.01325;
Ypa := ybar * 100000;


(*
Druck, Pascal Pa 1 Pa = 1 N/m2 = 1 kg/(s2 �E m) . 0,75 �E 10.2 mmHg
mechanische 1 MPa = 1 N/mm2 . fur Festigkeitsangaben
Spannung Bar bar 1 bar = 105 Pa = 103 mbar = 105 kg/(s2 �E m)
Millimeter- mmHg 1 mmHg = 133,322 Pa = 1,333 22 mbar
Quecksilbersaule . nur in Heilkunde zulassig
physik. Atmosphare atm 1 atm = 1,013 25 bar
techn. Atmosphare at 1 at = 1 kp/cm2 = 0,980665 bar
Torr Torr 1 Torr = (101325/760) Pa = 1,333224 mbar
Meter-Wassersaule mWS 1 mWS = 9806,65 Pa = 98,0665 mbar
psi lbf/in2 1 lbf/in2 = 68,947 57 mbar = 6894,757 Pa

*)
END_FUNCTION_BLOCK

(* POU BUFFER_COMP, ST *)
FUNCTION BUFFER_COMP : INT
VAR_INPUT
	PT1 : POINTER TO ARRAY[0..32767] OF BYTE;
	SIZE1 : INT;
	PT2 : POINTER TO ARRAY[0..32767] OF BYTE;
	SIZE2 : INT;
	START : INT;
END_VAR
VAR
	i, j, end : INT;
END_VAR

(*
version 1.0	14. nov. 2008
programmer 	hugo
tested by	oscat


 
*)
(* search for first character match *)
IF size2 <= size1 THEN
	end := size1 - size2;
	FOR i := START TO end DO
		IF PT1^[i] = PT2^[0] THEN
			(* first character matches, now compare rest of array *)
			j := 1;
			WHILE j < size2 DO
				IF pt2^[j] <> pt1^[j+i] THEN EXIT; END_IF;
				j := j + 1;
			END_WHILE;
			(* when J > size2 a match was found return the position i in buffer1 *)
			IF j = size2 THEN
				BUFFER_COMP := i;
				RETURN;
			END_IF;
		END_IF;
	END_FOR;
END_IF;
BUFFER_COMP := -1;


(*
hm 	14. nov. 2008	rev 1.0
	original version

*)
END_FUNCTION

(* POU BUFFER_SEARCH, ST *)
FUNCTION BUFFER_SEARCH : INT
VAR_INPUT
	PT : POINTER TO ARRAY[0..32767] OF BYTE;
	SIZE : UINT;
	STR : STRING(STRING_LENGTH);
	POS : INT;
	IGN : BYTE;
END_VAR
VAR
	ps : POINTER TO ARRAY[0..255] OF BYTE;
	i: INT;
	end: INT;
	k: INT;
	lx: INT;
END_VAR


(*
version 1.2	13. may. 2008
programmer 	hugo
tested by	oscat

this function will search for a string STR in an array of byte starting at position pos.
the function needs to be called:	buffer_search(adr("array"),sizeof("array"), STR, POS, IGN);
because this function works with pointers its very time efficient and it needs no extra memory.
The function returns the position of the first character of the string in the array if found.
a 0 is returned if the string is not found in the array.
The parameter IGN specifies a wildcard character in the search string.

*)
ps := ADR(str);
lx := LEN(str);
end := UINT_TO_INT(size) - lx;
lx := lx - 1;
FOR i := pos TO end DO
	FOR k := 0 TO lx DO
		IF (ps^[k] <> ign) AND (ps^[k] <> pt^[i+k]) THEN EXIT; END_IF;
	END_FOR;
	IF k > lx THEN
		BUFFER_SEARCH := i;
		RETURN;
	END_IF;
END_FOR;
BUFFER_SEARCH := 0;


(* revision History

hm 5. mar. 2008	rev 1.0
	original version

hm	16. mar. 2008	rev 1.1
	chaged type of input size to uint

hm	13. may. 2008	rev 1.2
	changed type of pointer to array[1..32767]
	changed size of string to STRING_LENGTH

*)
END_FUNCTION

(* POU BUFFER_TO_STRING, ST *)
FUNCTION BUFFER_TO_STRING : STRING(STRING_LENGTH)
VAR_INPUT
	PT : POINTER TO ARRAY[0..32767] OF BYTE;
	SIZE : UINT;
	START : UINT;
	STOP : UINT;
END_VAR
VAR
	ps : POINTER TO BYTE;
	i : INT;
END_VAR


(*
version 1.3	12. jun. 2008
programmer 	hugo
tested by	oscat

this function will retrieve a string from an array of byte starting at position start and stop at position stop.
the function needs to be called:	buffer_TO_String(adr("array"),sizeof("array"), start, stop);
because this function works with pointers its very time efficient and it needs no extra memory.

*)
ps := ADR(BUFFER_TO_STRING);
start :=MIN(start, size);
stop := MIN(stop, size);
(* check for maximum string_length *)
IF UINT_TO_INT(stop - start + 1) >= STRING_LENGTH THEN
	stop := start + INT_TO_UINT(STRING_LENGTH) - 1;
END_IF;

FOR i := UINT_TO_INT(start) TO UINT_TO_INT(stop) DO
	ps^ := pt^[i];
	ps := ps + 1;
END_FOR;

(* terminate the string *)
ps^ := 0;



(* revision History
hm 	5. mar. 2008	rev 1.0
	original version

hm	16. mar. 2008	rev 1.1
	changed type of input size to uint

hm	13. may. 2008	rev 1.2
	changed type of pointer to array[0..32767]
	changed size of string to STRING_LENGTH

hm	12. jun. 2008	rev 1.3
	check for pointer overrun
	change input start and stop to uint
	added type conversions to avoid warnings under codesys 3.0


*)
END_FUNCTION

(* POU BURNER, ST *)
FUNCTION_BLOCK BURNER
VAR_INPUT
	in : BOOL;
	stage2 : BOOL;
	over_temp : BOOL;
	oil_temp : BOOL := TRUE;
	Flame : BOOL;
	rst : BOOL;
	rst_timer : BOOL;
END_VAR
VAR_INPUT CONSTANT
	pre_heat_time : TIME := t#5s;
	pre_vent_time : TIME := t#15s;
	pre_ignite_time : TIME := t#5s;
	post_ignite_time : TIME := t#25s;
	stage2_delay : TIME := t#10s;
	safety_time : TIME := t#5s;
	lockout_time : TIME := t#10s;
	multiple_ignition : BOOL := TRUE;
	KW1 : REAL;
	KW2 : REAL;
END_VAR
VAR_OUTPUT
	motor : BOOL;
	coil1 : BOOL;
	coil2 : BOOL;
	pre_heat: BOOL;
	ignite : BOOL;
	KWh : REAL;
	status : BYTE;
	fail : BOOL;
END_VAR
VAR_IN_OUT
	runtime1 : UDINT;
	runtime2 : UDINT;
	cycles : UDINT;
END_VAR
VAR
	state : BYTE;
	last : TIME;
	tx: TIME;
	last_change: TIME;
	timer1 : ONTIME;
	timer2 : ONTIME;
	oil_temp_last: BOOL;
	cycles2 : UDINT;
END_VAR

(*
version 1.5	15 sep 2007
programmer 	oscat
tested by	oscat

burner ist eine Oel-Brenner_steuerung fuer nichtmodulierende Oelbrenner
die steuerung kann ueber setup werte programmiert werden und entsprechenden brennern angepasst werden.
die vorheizzeit ist die zeit die eine oelvorwaermung aufgeheizt wird bevor der motor gestartet wird.
der eingang oil_temp gibt an ob die oil_temp erreicht wurde, er ist default auf true und kann auch offen gelassen werden.
die vorbelueftungszeit ist die zeit die der luefter laeuft bevor die oelzufuhr freigegeben wird.
die vorzuendzeit iust diejenige zeit die die zuendung vor offnen des oelventiel gestartet wird.
nachzuendzeit ist die zeit die nach entzuendung der flamme noch gezuendet wird.
die sicherheitszeit ist die zeit nach der die oelzufuhr gesperrt wird wenn keine flamme entsteht.
nach ablauf der sicherheitszeit wird ein fehler flag gesetzt und kann erst nach der sperrzeit wieder durch einen reset geloescht werden.
waehrend der sperrzeit ist keine weitere zuendung oder einschalten moeglich.
das flag mehrfachzuendung gibt an ob eine erloschene flamme in betrieb automatisch wieder gezuendet werden soll.
der flammwaechster liegt auf eingang flamme, ein uebertemperaturschutz auf dem eingang over_temp
der betriebsstundenzaehler gibt die brennerstunden in stunden als real ausgabewer an.
der ausgang motor steuert den luefter / pumpenmotor, oil_ventil schaltet das oil ventil und zuendung schaltet die zuendung ein.

if output fail > 0 an error happened and the output has an error code:
0 :	no error
1 :	pre heating time expired and oil temp input is not true
2 :	flame monitor is active during preheating time
3 :	flame monitor active during pre_ventilation_time
4 :	no ignoition during safety time
5 :	no flame during operation
9 :	overtemp input is true

*)
(* read system time *)
tx := DWORD_TO_TIME(T_PLC_MS());

(* check rst input and overtemp *)
IF rst OR over_temp OR state = 0 THEN
	IF status > 0 AND tx - last_change >= lockout_time AND rst THEN
		status := 110;
		fail := FALSE;
		state := 1;
	ELSE
		(* normaler reset *)
		motor := FALSE;
		coil1 := FALSE;
		coil2 := FALSE;
		ignite := FALSE;
		pre_heat := FALSE;
		IF over_temp THEN
			status := 9;
			fail := TRUE;
		END_IF;
		last_change := tx;
		last := tx;
		state := 1;
	END_IF;
END_IF;

(* check for timer rst and rst timer if true *)
IF rst_timer THEN
	runtime1 := 0;
	runtime2 := 0;
	cycles := 0;
	cycles2 := 0;
END_IF;

(* quit here if an error is present *)
IF (status > 0 AND status < 100) OR rst THEN RETURN; END_IF;

(* start sequence *)
CASE state OF

1:	(* in signal starts oil pre heating *)
	IF in AND flame THEN
		state := 7;
		pre_heat := FALSE;
		status := 2;
		last_change := tx;
	ELSIF in THEN
		pre_heat := TRUE;
		state := 2;
		last_change := tx;
	END_IF;

2:	(* after pre_heating time start motor *)
	IF (tx- last_change >= pre_heat_time AND oil_temp) OR (oil_temp AND NOT oil_temp_last) THEN
		motor := TRUE;
		state := 3;
		last_change := tx;
	(* pre_heat_time ist abgelaufen und oil_temp ist nicht aktiv *)
	ELSIF tx - last_change >= pre_heat_time AND NOT oil_temp THEN
		state := 7;
		pre_heat := FALSE;
		status := 1;
		last_change := tx;
	(* flame monitor cannot be active at this time *)
	ELSIF flame THEN
		state := 7;
		pre_heat := FALSE;
		status := 2;
		last_change := tx;
	END_IF;

3:	(* abwarten bis zündung eingeschaltet werden kann *)
	IF tx - last_change >= pre_vent_time - pre_ignite_time THEN
		ignite := TRUE;
		state := 4;
		last_change := tx;
	(* flame monitor cannot be active at this time *)
	ELSIF flame THEN
		state := 7;
		pre_heat := FALSE;
		motor := FALSE;
		status := 3;
		last_change := tx;
	END_IF;

4:	(* warten bis oelzufuhr geoeffnet werden darf *)
	IF tx - last_change >= pre_ignite_time THEN
		coil1 := TRUE;
		state := 5;
		last_change := tx;
	END_IF;

5:	(* warten auf flammwaechter und falls noetig abschalten *)
	IF tx - last_change >= safety_time OR flame THEN
		IF NOT flame THEN
			(* notabschaltung da flammwaechster nicht angesprochen hat *)
			state := 7;
			motor := FALSE;
			coil1 := FALSE;
			pre_heat := FALSE;
			ignite := FALSE;
			status := 4;
			last_change := tx;
		ELSE
			state := 6;
			last_change := tx;
		END_IF;
	END_IF;

6:	(* brenner läuft, flammueberwachung und nach ablauf der nachigniteszeit ignite abschalten *)
	IF NOT flame AND NOT multiple_ignition THEN
		(* notabschaltung da flammwaechster keine flamme meldet *)
		state := 7;
		motor := FALSE;
		coil1 := FALSE;
		coil2 := FALSE;
		pre_heat := FALSE;
		ignite := FALSE;
		status := 5;
		last_change := tx;
	ELSIF NOT flame AND multiple_ignition THEN
		ignite := TRUE;
		state := 5;
		coil2 := FALSE;
		last_change := tx;
	ELSE
		IF tx - last_change >= post_ignite_time THEN
			(* post_ignite_time abgelaufen, ignite abschalten *)
			ignite := FALSE;
		END_IF;
		IF tx - last_change >= stage2_delay AND stage2 THEN
			coil2 := TRUE;
		ELSE
			coil2 := FALSE;
		END_IF;
	END_IF;
END_CASE;

(* abschaltung wenn kein eingangssignal *)
IF NOT in THEN
	state := 1;
	motor := FALSE;
	coil1 := FALSE;
	coil2 := FALSE;
	ignite := FALSE;
	pre_heat := FALSE;
	last_change := tx;
END_IF;

(* runtimezähler *)
timer1(in := flame AND in AND motor AND coil1 AND NOT coil2, seconds := runtime1, cycles := cycles);
timer2(in := flame AND in AND motor AND coil1 AND coil2, seconds := runtime2, cycles := cycles2);
KWH := UDINT_TO_REAL(runtime1) * KW1 / 3600.0 + UDINT_TO_REAL(runtime2) * KW2 / 3600.0;

(* zeit fuer naechsten aufruf merken *)
last := tx;

(* set fail output IF ERROR and Status  if normal operation *)

IF status > 0 AND status < 100 THEN
	fail := TRUE;
ELSE
	fail := FALSE;
	IF NOT in THEN
		status := 110;
	ELSIF flame AND in AND motor AND coil2 AND coil1 THEN
		status := 113;
	ELSIF flame AND in AND motor AND coil1 THEN
		status := 112;
	ELSE
		status := 111;
	END_IF;
END_IF;



(*
31.12.2006	hm		rev 1.1
	added pre_heat timing and output
	flame monitor before ignition will generate error on status output
	added output for KWh

31.12.2006	hm		rev 1.2
	added oil_temp_input

31.12.2006	hm		rev 1.3
	changed status output to be byte instead of bool

22.1.2007		hm		rev 1.4
	renamed fail output to status
	added output cycles
	corrected an error while pre_heat would be on when an error was present
	added coil2 output and stage2 input

15.9.2007		hm		rev 1.5
	replaced Time() with T_PLC_MS for compatibility and performance reasons

hm	21. oct. 2008	rev 1.6
	changed code to use new ontime rev 2.0	
*)
END_FUNCTION_BLOCK

(* POU BYTE_OF_BIT, ST *)
FUNCTION BYTE_OF_BIT : BYTE
VAR_INPUT
	B0:BOOL;
	B1:BOOL;
	B2:BOOL;
	B3:BOOL;
	B4:BOOL;
	B5:BOOL;
	B6:BOOL;
	B7:BOOL;
END_VAR
VAR
END_VAR

(*
version 1.1	 18. feb 2006
programmer 	hugo
tested by		tobias

this function creates a byte from 8 individual bits

*)
Byte_of_bit := SHL(SHL(SHL(SHL(SHL(SHL(SHL(BOOL_TO_BYTE(B7),1) OR BOOL_TO_BYTE(B6),1) OR BOOL_TO_BYTE(B5),1) OR BOOL_TO_BYTE(B4),1)
	OR BOOL_TO_BYTE(B3),1) OR BOOL_TO_BYTE(B2),1) OR BOOL_TO_BYTE(B1),1) OR BOOL_TO_BYTE(B0);


(* revision history

hm	4. aug 2006		rev 1.0
	original version

hm	18. feb. 2008	rev 1.1
	improved performance

*)
END_FUNCTION

(* POU BYTE_OF_DWORD, ST *)
FUNCTION BYTE_OF_DWORD : BYTE
VAR_INPUT
	in : DWORD;
	N : BYTE;
END_VAR
VAR
END_VAR

(*
version 1.2	30. oct. 2008
programmer 	hugo
tested by	oscat

this function extracts a single byte from the nth position from right (right is lowest byte) 
the lower byte (starting with Bit0 from in) is selected with N=0.
*)
BYTE_OF_DWORD := DWORD_TO_BYTE(SHR(in,SHL(n,3)));

(* revision history
hm	17. jan 2007	rev 1.0
	original version

hm	2. jan 2008		rev 1.1
	improved performance

hm	30. oct. 2008	rev 1.2
	improved performance
*)
END_FUNCTION

(* POU BYTE_TO_BITS, ST *)
FUNCTION_BLOCK BYTE_TO_BITS
VAR_INPUT
	IN: BYTE;
END_VAR
VAR_OUTPUT
	B0: BOOL;
	B1: BOOL;
	B2: BOOL;
	B3: BOOL;
	B4: BOOL;
	B5: BOOL;
	B6: BOOL;
	B7: BOOL;
END_VAR
VAR
END_VAR

(*
version 1.1	16. mar. 2008
programmer 	hugo
tested by		tobias

this Function Block extracts the 8 Bits from a byte


*)
B0 := IN.0;
B1 := IN.1;
B2 := IN.2;
B3 := IN.3;
B4 := IN.4;
B5 := IN.5;
B6 := IN.6;
B7 := IN.7;

(* revision history
hm		4. aug 2006	rev 1.0
	original version

hm		16. mar 2008	rev 1.1
	renamed from byte_to_bit to byte_to_bits for compatibility reasons

*)
END_FUNCTION_BLOCK

(* POU BYTE_TO_RANGE, ST *)
FUNCTION BYTE_TO_RANGE : REAL
VAR_INPUT
	X : BYTE;
	low : REAL;
	high : REAL;
END_VAR
VAR
END_VAR

(*
version 1.0	9. jan 2008
programmer 	hugo
tested by		tobias

Byte_to_Range converts a Byte into a real between low and high.

*)
Byte_to_Range := (high - low) * X / 255.0 + low;


(* revision history
hm	9. jan 2008		rev 1.0
	original version

*)
END_FUNCTION

(* POU BYTE_TO_STRB, ST *)
FUNCTION BYTE_TO_STRB : STRING(8)
VAR_INPUT
	IN : BYTE;
END_VAR
VAR
	i: INT;
	pt : POINTER TO BYTE;
END_VAR

(*
version 1.3	20. jun. 2008
programmer 	hugo
tested by	oscat

BYTE_TO_STRINGB converts a Byte to a String of Bits represented by '0' and '1' s.
The lowest order bit will be on the right and the high order bit on the left.

*)
(* pointer für die ausgabe ermitteln *)
pt := ADR(BYTE_TO_STRB);
(* die 8 ausgabecharacter ermitteln und schreiben *)
FOR i := 1 TO 8 DO
	pt^ := BOOL_TO_BYTE(in.7) + 48;
	in := SHL(in,1);
	pt := pt + 1;
END_FOR;

(* der ausgabestring muss noch mit 0 abgeschlossen werden *)
pt^ := 0;

(* code before rev 1.1
FOR i := 1 TO 8 DO
	IF in.0 = 0 THEN temp := CONCAT('0', temp); ELSE temp := CONCAT('1', temp); END_IF;
	in := SHR(in, 1);
END_FOR;
BYTE_TO_STRB := temp;
*)


(* revision history

hm		9.6.2007	rev 1.0		
	original version 

hm	15. dec 2007	rev 1.1
	inprooved code for higher performance

hm	29. mar. 2008	rev 1.2
	changed STRING to STRING(8)

hm	20. jun. 2008	rev 1.3
	performance improvement

*)
END_FUNCTION

(* POU BYTE_TO_STRH, ST *)
FUNCTION BYTE_TO_STRH : STRING(2)
VAR_INPUT
	IN : BYTE;
END_VAR
VAR
	temp : BYTE;
	PT : POINTER TO BYTE;
END_VAR

(*
version 1.3	29 mar. 2008
programmer 	hugo
tested by		tobias

BYTE_TO_STRINGH converts a Byte to a String of Hexadecimal represented by '0' .. '9' and 'A' .. 'F'.
The lowest order Character will be on the right and the high order Character on the left.

*)
(* read pointer to output string *)
PT := ADR(BYTE_TO_STRH);
(* calculate high order hex value *)
temp := SHR(in,4);
(* convert value to hex character *)
IF temp <= 9 THEN temp := temp + 48; ELSE temp := temp + 55; END_IF;
(* write friat character to output string *)
PT^ := temp;
(* calculate low order hex value *)
temp := in AND 2#00001111;
IF temp <= 9 THEN temp := temp + 48; ELSE temp := temp + 55; END_IF;
(* increment pointer and wirte low order character *)
pt := pt + 1;
pt^ := temp;
(* set pointer at the end of the output string and close the string with 0 *)
pt := pt + 1;
pt^:= 0;


(* code before rev 1.2
FOR i := 1 TO 2 DO
	X := in AND 2#1111;
	IF X <= 9 THEN X := X + 48; ELSE X := X + 55; END_IF;
	Cx := CHR(X);
	temp := CONCAT(Cx, temp);
	in := SHR(in,4);
END_FOR;
BYTE_TO_STRH := temp;
*)

(* revision history

hm	9.6.2007		rev 1.0		
	original version 

hm	11.9.2007		rev 1.1		
	changed coding for compatibility with twincat, under twincat concat cannot have a function as argument.	

hm	15 dec 2007		REV 1.2
	changed code for higher performance

hm	29. mar. 2008	rev 1.3
	changed STRING to STRING(2)
*)
END_FUNCTION

(* POU C_TO_F, ST *)
FUNCTION C_TO_F : REAL
VAR_INPUT
	celsius : REAL;
END_VAR
VAR
END_VAR

(*
version 1.0	4 aug 2006
programmer 	hugo
tested by		tobias

this function converts celsius  to fahrenheit 

*)
C_to_F := celsius * 1.8 + 32;
END_FUNCTION

(* POU C_TO_K, ST *)
FUNCTION C_TO_K : REAL
VAR_INPUT
	Celsius : REAL;
END_VAR
VAR
END_VAR

(*
version 1.0	4 dec 2006
programmer 	hugo
tested by		tobias

this function converts celsius to kelvin
*)
C_to_K := Celsius - 273.15;
END_FUNCTION

(* POU CABS, ST *)
FUNCTION CABS : REAL
VAR_INPUT
	X : complex;
END_VAR
VAR
END_VAR

(*
version 1.0	21 feb 2008
programmer 	hugo
tested by	oscat

this function the aboslute value of a complex number

*)
CABS := HYPOT(x.re, x.im);


(* revision history
hm	21. feb 2008	rev 1.0
	original version

*)
END_FUNCTION

(* POU HYPOT, ST *)
FUNCTION HYPOT : REAL
VAR_INPUT
	X : REAL;
	Y : REAL;
END_VAR
VAR
END_VAR

(*
version 1.0	21 feb 2008
programmer 	hugo
tested by	oscat

this function calculates the pythagorean function

*)
HYPOT := SQRT(x*x + y*y);


(* revision history
hm	21. feb 2008	rev 1.0
	original version

*)
END_FUNCTION

(* POU CACOS, ST *)
FUNCTION CACOS : complex
VAR_INPUT
	X : complex;
END_VAR
VAR
	Y : complex;
END_VAR

(*
version 1.0	21 feb 2008
programmer 	hugo
tested by	oscat

this function calculates the arcus cosinus function of a complex number

*)
y := CACOSH(x);
CACOS.re := y.im;
CACOS.im := -y.re;



(* revision history
hm	21. feb 2008	rev 1.0
	original version


*)
END_FUNCTION

(* POU CACOSH, ST *)
FUNCTION CACOSH : complex
VAR_INPUT
	X : complex;
END_VAR
VAR
	Y : complex;
END_VAR

(*
version 1.0	21 feb 2008
programmer 	hugo
tested by	oscat

this function calculates the hyperbolic arcus cosinus function of a complex number

*)
y.re := (X.re - X.im)*(X.re + X.im) - 1.0;
y.im := 2.0 * X.re * X.im;
y    := CSQRT(y);
y.re := y.re + x.re;
y.im := y.im + x.im;
CACOSH  := CLOG(y);



(* revision history
hm	21. feb 2008	rev 1.0
	original version


*)
END_FUNCTION

(* POU CSQRT, ST *)
FUNCTION CSQRT : complex
VAR_INPUT
	X : complex;
END_VAR
VAR
	temp : REAL;
END_VAR

(*
version 1.0	21 feb 2008
programmer 	hugo
tested by	oscat

this function calculates the complex sqare root

*)
temp := HYPOT(x.re, x.im);
CSQRT.re :=  SQRT(0.5 * (temp + x.re));
CSQRT.im :=  sgn(x.im) * SQRT(0.5 * (temp - x.re));


(* revision history
hm	21. feb 2008	rev 1.0
	original version

*)
END_FUNCTION

(* POU SGN, ST *)
FUNCTION SGN : INT
VAR_INPUT
	X : REAL;
END_VAR
VAR
END_VAR

(*
version 1.1	11. nov. 2008
programmer 	hugo
tested by	tobias

sgn returns 0 when X = 0 , -1 when X < 1 and +1 when X > 1

*)
IF X > 0 THEN
	SGN := 1;
ELSIF X < 0 THEN
	SGN := -1;
ELSE
	SGN := 0;
END_IF;



(* revision histroy
hm	16. oct 2007	rev 1.0
	original version

hm	11. nov 2007	rev 1.1
	changed type of function from real to int

*)
END_FUNCTION

(* POU CLOG, ST *)
FUNCTION CLOG : complex
VAR_INPUT
	X : complex;
END_VAR
VAR
END_VAR

(*
version 1.1	20. apr. 2008
programmer 	hugo
tested by	oscat

this function calculates the complex natural (base e) logarithm

*)
CLOG.re := LN(HYPOT(X.re, X.im));
CLOG.im := ATAN2(X.im, X.re);


(* revision history
hm	21. feb 2008	rev 1.0
	original version

hm	20. apr. 2008	rev 1.1
	use ATAN2 instead of ATAN
*)
END_FUNCTION

(* POU CADD, ST *)
FUNCTION CADD : complex
VAR_INPUT
	X, Y : complex;
END_VAR
VAR
END_VAR

(*
version 1.0	21 feb 2008
programmer 	hugo
tested by	oscat

this function add two complex numbers

*)
CADD.re := x.re + y.re;
CADD.im := x.im + y.im;


(* revision history
hm	21. feb 2008	rev 1.0
	original version

*)
END_FUNCTION

(* POU CALENDAR_CALC, ST *)
FUNCTION_BLOCK CALENDAR_CALC
VAR_INPUT
END_VAR
VAR_IN_OUT
	XCAL : CALENDAR;
END_VAR
VAR
	last : DT;
	last_day : DINT;
	holy : HOLIDAY;
	sun : SUN_TIME;
	last_hour: INT;
	utod: TOD;
	pos : SUN_POS;
END_VAR
VAR_TEMP
	dtemp : DINT;
	tmp : INT;
END_VAR


(*
version 1.1	8. feb. 2009
programmer 	hugo
tested by		oscat

calendar calc liest die weltzeit .UTC aus einer CALENDAR Struktur und berechnet die restlichen Werte der Struktur
calendar_calc stellt sicher das die Werte fortlaufend aktualisiert werden und dabei funktionen nur dann aufgerufen werden wenn dies nötig ist.

*)
IF xcal.UTC <> last THEN
	(* run once per second *)
	last := XCAL.UTC;
	utod := DT_TO_TOD(xcal.UTC);
	(* calculate ltc from utc *)
	XCAL.LDT := UTC_TO_LTIME(XCAL.UTC, XCAL.DST_EN, XCAL.OFFSET);
	XCAL.LDATE := DT_TO_DATE(XCAL.LDT);
	XCAL.LTOD := DT_TO_TOD(XCAL.LDT);
	dtemp := DAY_OF_DATE(XCAL.LDATE);
	IF dtemp <> last_day THEN
		last_day := dtemp;
		(* a new day has started, recalculate daily events *)
		XCAL.YEAR := YEAR_OF_DATE(XCAL.LDATE);
		XCAL.MONTH := MONTH_OF_DATE(XCAL.LDATE);
		XCAL.DAY := DAY_OF_MONTH(XCAL.LDATE);
		XCAL.WEEKDAY := DAY_OF_WEEK(XCAL.LDATE);
		HOLY(date_in := XCAL.LDATE, country := XCAl.LOCATION);
		XCAL.HOLIDAY := HOLY.Y;
		XCAL.HOLY_NAME := HOLY.NAME;
		sun(latitude := XCAL.LATITUDE, longitude := xcal.LONGITUDE, utc := xcal.UTC);
		XCAL.SUN_RISE := sun.sun_rise;
		XCAL.SUN_SET := sun.sun_set;
	END_IF;
	tmp := HOUR(xcal.LTOD);
	IF  tmp <> last_hour THEN
		XCAL.DST_ON := DST(XCAL.UTC);
		last_hour := tmp;
	END_IF;
	xcal.night := utod < xcal.SUN_RISE OR utod > xcal.SUN_SET;
	(* calculate the suns position *)
	pos(latitude := xcal.LATITUDE, longitude := xcal.LONGITUDE, utc := xcal.UTC);
	xcal.SUN_HOR := pos.B;
	xcal.SUN_VER := pos.HR;
END_IF;



(* revision history

hm 23. oct. 2008	rev 1.0
	original version

hm	8. feb. 2009	rev 1.1
	night was calculated wrong
	added sun position data
	
*)
END_FUNCTION_BLOCK

(* POU HOLIDAY, ST *)
FUNCTION_BLOCK HOLIDAY
VAR_INPUT
	DATE_IN : DATE;
	COUNTRY : INT;
	FRIDAY : BOOL;
	SATURDAY : BOOL;
	SUNDAY : BOOL;
END_VAR

VAR CONSTANT
	SIZE : INT := 29;
END_VAR
VAR_OUTPUT
	Y : BOOL;
	NAME : STRING(30);
END_VAR
VAR
	last_active : DATE;
	ostern: DATE;
	i: INT;
	jahr: INT;
	x_date: DATE;
	cx: INT;
	wdx: INT;
	check: HOLIDAY_DATA;
END_VAR

(*
version 1.6	21. oct. 2008
programmer 	hugo
tested by	tobias

holiday calculates if a given day is a holiday and displays the name of the holiday as string as well as a boolean flag to indicate a holiday.
the holidays are specified in the country setup under global constants.
a holiday can be of fixed date for example new years day on january 1st.
a holiday can have a fixed offset from easter sunday as for most church holidays.
a holiday can be a specific weekday before a fixed date, for example buss und bettag is the last wednesday before nov 23rd.
with a simple f_use flag any specific holiday can be turned on or off if needed.

*)
(* for performance reasons only activate once a day *)
IF last_active = date_in THEN RETURN; END_IF;

(* determine country *)
IF COUNTRY = 0 THEN
	cx := location.DEFAULT;
ELSE
	cx := MIN(location.LMAX, COUNTRY);
END_IF;

(* berechnung von ostern für das aktuelle jahr *)
jahr := YEAR_OF_DATE(date_in);
ostern := EASTER(jahr);
last_active := DATE_IN;
wdx := DAY_OF_WEEK(DATE_IN);

(* check array if today is holiday *)
Y := (wdx = 5 AND FRIDAY) OR (wdx = 6 AND SATURDAY) OR (wdx = 7 AND SUNDAY);
NAME := '';

FOR i := 0 TO size DO
	check := location.HOLIDAY[cx, i];
	x_date := SET_DATE(jahr, check.MONTH , check.DAY);
	IF check.USE = 1 AND check.MONTH > 0 THEN
		(* check for fixed date holiday *)
		IF x_date = date_in THEN
			Y := TRUE;
			NAME := check.NAME;
			RETURN;
		END_IF;
	ELSIF check.USE = 1 AND check.MONTH = 0 THEN
		(* check for holiday in reference to easter *)
		IF DATE_ADD(ostern, check.DAY ,0,0,0) = date_in THEN
			Y := TRUE;
			NAME := check.NAME;
			RETURN;
		END_IF;
	ELSIF check.USE < 0 THEN
		(* check for holiday on a weekday before date *)
		IF DAY_OF_WEEK(date_in) = ABS(check.USE) AND date_in < x_date AND date_in >= DATE_ADD(x_date,-7,0,0,0) THEN
			Y := TRUE;
			NAME := check.NAME;
			RETURN;
		END_IF;
	END_IF;
END_FOR;



(*
Neujahrstag 	1. Januar 	• 	• 	• 	• 	• 	• 	• 	• 	• 	• 	• 	• 	• 	• 	• 	•
Heilige Drei Könige 	6. Januar 	• 	• 												• 		
Karfreitag 	Ostersonntag - 2d 	• 	• 	• 	• 	• 	• 	• 	• 	• 	• 	• 	• 	• 	• 	• 	•
Ostersonntag 	siehe Osterdatum 				(•) 												
Ostermontag 	Ostersonntag + 1d 	• 	• 	• 	• 	• 	• 	• 	• 	• 	• 	• 	• 	• 	• 	• 	•
Tag der Arbeit 	1. Mai 	• 	• 	• 	• 	• 	• 	• 	• 	• 	• 	• 	• 	• 	• 	• 	•
Christi Himmelfahrt 	Ostersonntag + 39d 	• 	• 	• 	• 	• 	• 	• 	• 	• 	• 	• 	• 	• 	• 	• 	•
Pfingstsonntag 	Ostersonntag + 49d 				(•) 												
Pfingstmontag 	Ostersonntag + 50d 	• 	• 	• 	• 	• 	• 	• 	• 	• 	• 	• 	• 	• 	• 	• 	•
Fronleichnam 	Ostersonntag + 60d 	• 	• 					• 			• 	• 	• 	1) 			2)
Augsburger Friedensfest 	8. August 		(3) 														
Mariä Himmelfahrt 	15. August 		(5) 										• 				
Tag der Deutschen Einheit 	3. Oktober 6) 	• 	• 	• 	• 	• 	• 	• 	• 	• 	• 	• 	• 	• 	• 	• 	•
Reformationstag 	31. Oktober 				• 				• 					• 	• 		•
Allerheiligen 	1. November 	• 	• 								• 	• 	• 				
Buß- und Bettag 4) 	Mittwoch vor dem 23.11. 			7 										• 			
1. Weihnachtstag 	25. Dezember 	• 	• 	• 	• 	• 	• 	• 	• 	• 	• 	• 	• 	• 	• 	• 	•
2. Weihnachtstag 	26. Dezember 	• 	• 	• 	• 	• 	• 	• 	• 	• 	• 	• 	• 	• 	• 	• 	•
*)



(* revision history
hm 	27. feb. 2007	rev 1.1
	deleted unused variable init

hm	31. oct. 2007	rev 1.2
	changed holiday definition from constant to input constant to allow easier changes by user without recompilation of the lib

hm 	24. nov. 2007	rev 1.3
	changes F_use of  Buß_und_Bettag to 0 because this is no official holiday

hm	7. apr. 2008	rev 1.4
	improved performance

hm	7. oct. 2008	rev 1.5
	changed code to use setup data from global constants
	changed length of output NAME from 20 to 30
	holiday will now also be indicated on a weekend
	changed function year to year_of_date
	changed function weekday to day_of_week

hm	21. oct. 2008	rev 1.6
	using location constants
*)
END_FUNCTION_BLOCK

(* POU YEAR_OF_DATE, ST *)
FUNCTION YEAR_OF_DATE : INT
VAR_INPUT
	IDATE : DATE;
END_VAR
VAR
END_VAR

(*
version 1.4	7. oct. 2008
programmer 	hugo
tested by	oscat

returs the year of a date  
the function works for dates from 1970 - 2099 

*)
YEAR_OF_DATE := DWORD_TO_INT((DATE_TO_DWORD(idate)+43200) / 31557600 + 1970);


(* code used prior to rev 1.1
year := DWORD_TO_INT((DATE_TO_DWORD(idate)/864+71954300)/36525);
*)

(* revision history
hm	4. aug 2006		rev 1.0
	original version

hm	1. okt 2007		rev 1.1
	corrected error in algorithm
	adjustment for S7 compatibility

hm	23.12.2007		rev 1.2
	changed code for better performance

hm	7. apr. 2008	rev 1.3
	deleted unused step7 code

hm	7. oct. 2008	rev 1.4
	reneamed function (year) to year_of_date

*)
END_FUNCTION

(* POU EASTER, ST *)
FUNCTION EASTER : DATE
VAR_INPUT
	year : INT;
END_VAR
VAR
	b,c: INT;
	oday: INT;
END_VAR

(*
version 1.3	7. apr. 2008
programmer 	hugo
tested by	tobias

easter calculates the day of easter sunday for a given year.
most other catholic holidays are calculated in reference to easter sunday.

*)
b := (204 - 11 * (YEAR MOD 19)) MOD 30;
IF b > 27 THEN b := b - 1; END_IF;
c := (year + SHR(year,2) + b - 13) MOD 7;
oday := 28 + b - c;
IF oday > 33 THEN
	easter := set_Date(year, 4, oday - 31);
ELSE
	EASTER := SET_DATE(year, 3, oday);
END_IF;




(* alternativer algorithmus ueber das pasah fest
execution time roughly 200us
Der sog. Passah-Vollmond wird berechnet, in dem das Jahr durch 19 ge-
teilt wird und der Rest mit der folgenden Tabelle verglichen wird:
 
    0: Apr 14       5: Apr 18      10: Mrz 25      15: Mrz 30
    1: Apr 03       6: Apr 08      11: Apr 13      16: Apr 17
    2: Mrz 23       7: Mrz 28      12: Apr 02      17: Apr 07
    3: Apr 11       8: Apr 16      13: Mrz 22      18: Mrz 27
    4: Mrz 31       9: Apr 05      14: Apr 10
 
Faellt dieses Datum auf einen Sonntag, ist Ostern der naechste Sonntag!
 
Beispiel: 1992 MOD 19 = 16, daraus folgt 17.04., der naechste Sonntag
          ist dann der 19. April (Ostersonntag)
*)


(* this algorithm is 180 us
a := year MOD 19;
b := year / 100;
c := year MOD 100;
d := b / 4;
e := b MOD 4;
f := (b + 8) / 25;
g := (b - f + 1) / 3;
h := (19 * a + b - d -g + 15) MOD 30;
i := C / 4;
k := c MOD 4;
l := (32 + 2*e + 2*i - h - k) MOD 7;
m := (a + 11 * h + 22 * l) / 451;
x := h + l - 7 * m + 114;
n := X / 31;
o := x MOD 31 + 1;

easter := set_Date(year,n,o);
*)
(*
Im Magazin "Nature" vom 20. April 1876 veröffentlichte ein anonymer Autor eine Tabelle mit Regeln zur Berechnung des (Gregorianischen) Ostersonntages des Jahres J. In Formeln ausgedrückt erhält man das Folgende:
a	=	J mod 19
b	=	int(J / 100)
c	=	J mod 100
d	=	int(b / 4)
e	=	b mod 4
f	=	int((b + 8) / 25)
g	=	int((b - f + 1) / 3
h	=	(19 · a + b - d - g + 15) mod 30
i	=	int(c / 4)
k	=	c mod 4
l	=	(32 + 2 · e + 2 · i - h - k) mod 7
m	=	int((a + 11 · h + 22 · l) / 451)
n	=	int((h + l - 7 · m + 114) / 31)
o	=	(h + l - 7 · m + 114) mod 31

n ist hierbei die Nummer des Monats, o + 1 die Nummer des Tages auf welchen der Ostersonntag im Jahr J fällt. Dieser Algorithmus kommt ohne Hilfszahlen aus.

*)

(* revision history
hm	27. dec 2006	rev 1.0
	original version

hm	15. dec 2007	rev 1.1
	modified code for better performance

hm	3. feb 2008		rev 1.2
	modified code for better performance

hm	7. apr. 2008	rev 1.3
	improved performance
*)
END_FUNCTION

(* POU SET_DATE, ST *)
FUNCTION SET_DATE : DATE
VAR_INPUT
	YEAR : INT;
	MONTH : INT;
	DAY : INT;
END_VAR
VAR
	count : DWORD;
END_VAR

(*
version 2.1	16. nov. 2008
programmer 	hugo
tested by	tobias

creates a date output from year, month and day of month   

*)
(* calculate the amount of days to 31.12. the year before *)
count := SHR(INT_TO_DWORD(year) * 1461 - 2878173,2)+INT_TO_DWORD(day);
(* add the days for the month of the year *)
count := count + INT_TO_DWORD(setup.MTH_OFS[LIMIT(1,month,12)]);
(* for leap years and month > february then add one more day *)
IF month > 2 AND LEAP_YEAR(year) THEN count := count + 1; END_IF;
(* generate the date *)
SET_DATE := DWORD_TO_DATE(count * 86400);







(* revision history
hm	4. aug. 2006	rev 1.0
	original version

hm	19 sep. 2007	rev 1.1
	use function leap_year to calculate leap year, more exceptions are handled

hm	1. okt	2007	rev 1.2
	added compatibility to step7

hm	16.dec 2007		rev 1.3
	changed code to improove performance

hm	3. jan. 2008	rev 1.4
	further improvements in performance

hm	16. mar. 2008	rev 1.5
	added type conversions to avoid warnings under codesys 3.0

hm	7. apr. 2008	rev 1.6
	deleted unused step7 code

hm	14. oct. 2008	rev 1.7
	optimized code for better performance

hm	25. oct. 2008	rev 2.0
	new code using setup constants

hm	16. nov. 2008	rev 2.1
	added typecats to avoid warnings
*)
END_FUNCTION

(* POU LEAP_YEAR, ST *)
FUNCTION LEAP_YEAR : BOOL
VAR_INPUT
	yr : INT;
END_VAR
VAR
END_VAR

(*
version 1.1	2 oct 2006
programmer 	hugo
tested by		tobias


leap_year is true if the tested year is a leap year  
  
*)
leap_year := SHL(yr,14) = 0;

(* this code was used prior to rev 1.1

IF yr MOD 400 = 0 THEN leap_year := TRUE;
ELSIF yr MOD 100 = 0 THEN leap_year := FALSE;
ELSIF yr MOD 4 =0 THEN leap_year := TRUE;
ELSE leap_year := FALSE;
END_IF;

*)

(* change history

hm 	2.10.2006		rev 1.1
	the function now works for any year from 1970 up to 2100

hm	1. oct 2007		rev 1.2
	chaged code for higher performance
*)
END_FUNCTION

(* POU DAY_OF_WEEK, ST *)
FUNCTION DAY_OF_WEEK : INT
VAR_INPUT
	IDATE : DATE;
END_VAR
VAR
END_VAR

(*
version 1.4	7. oct. 2008
programmer 	hugo
tested by	tobias

calculates the weekday of a week according to ISO8601   
monday = 1 ..... sunday = 7  

*)
DAY_OF_WEEK := DWORD_TO_INT((DATE_TO_DWORD(idate)/86400+3) MOD 7) + 1;



(* revision history
hm 	21.8.06 		rev 1.1
	corrected a miscalculation

hm	23.12.2007		rev 1.2
	correction for step7

hm	7. apr. 2008	rev 1.3
	deleted unused step7 code

hm	7. oct. 2008	rev 1.4
	changed name of function from weekday to day_of_week

*)
END_FUNCTION

(* POU DATE_ADD, ST *)
FUNCTION DATE_ADD : DATE
VAR_INPUT
	IDATE : DATE;
	D : INT;
	W : INT;
	M : INT;
	Y : INT;
END_VAR
VAR
	mo: INT;
	yr : INT;
END_VAR


(*
version 1.4	7. oct 2008
programmer 	hugo
tested by	oscat

date_add adds days, weeks, month or years to a date.
negative inputs are allowed for subtraction.

*)
DATE_ADD := DWORD_TO_DATE(DATE_TO_DWORD(idate) + 86400 * INT_TO_DWORD(d) + 604800 * INT_TO_DWORD(w));
mo := MONTH_OF_DATE(DATE_ADD);
yr := YEAR_OF_DATE(DATE_ADD) + y + FLOOR(INT_TO_REAL(mo + m - 1) / 12.0);
mo := mo + (ABS(m) MOD 12) * SGN(m);
IF mo < 1 THEN
	mo := mo + 12;
ELSIF mo > 12 THEN
	mo := mo - 12;
END_IF;
DATE_ADD := SET_DATE(yr,mo,DAY_OF_MONTH(DATE_ADD));



(* revision history

hm 27.12.2006		rev 1.0

hm 12.4.2007		rev 1.1
	corrected an error while date would be incorrect when year  = 0

hm	1.11.2007		rev 1.2
	added int_to_dword stetements to avoid possible overrun with möller ecp4

hm	22. mar. 2008	rev 1.3
	fixed some bugs when month was negative

hm	7. oct. 2008	rev 1.4
	changed function year to year_of_date
	changed function month to month_of_date

*)
END_FUNCTION

(* POU MONTH_OF_DATE, ST *)
FUNCTION MONTH_OF_DATE : INT
VAR_INPUT
	IDATE : DATE;
END_VAR
VAR
END_VAR

(*
version 1.2	7. oct. 2008
programmer 	hugo
tested by	tobias

returns the month of the year

*)
MONTH_OF_DATE := DAY_OF_YEAR(IDATE);
IF LEAP_OF_DATE(IDATE) THEN
	CASE MONTH_OF_DATE OF
		1..31 	:	MONTH_OF_DATE := 1;
		32..60	:	MONTH_OF_DATE := 2;
		61..91	:	MONTH_OF_DATE := 3;
		92..121 :	MONTH_OF_DATE := 4;
		122..152:	MONTH_OF_DATE := 5;
		153..182:	MONTH_OF_DATE := 6;
		183..213:	MONTH_OF_DATE := 7;
		214..244:	MONTH_OF_DATE := 8;
		245..274:	MONTH_OF_DATE := 9;
		275..305:	MONTH_OF_DATE := 10;
		306..335:	MONTH_OF_DATE := 11;
		336..366:	MONTH_OF_DATE := 12;
	END_CASE;
ELSE
	CASE MONTH_OF_DATE OF
		1..31 	:	MONTH_OF_DATE := 1;
		32..59	:	MONTH_OF_DATE := 2;
		60..90	:	MONTH_OF_DATE := 3;
		91..120 :	MONTH_OF_DATE := 4;
		121..151:	MONTH_OF_DATE := 5;
		152..181:	MONTH_OF_DATE := 6;
		182..212:	MONTH_OF_DATE := 7;
		213..243:	MONTH_OF_DATE := 8;
		244..273:	MONTH_OF_DATE := 9;
		274..304:	MONTH_OF_DATE := 10;
		305..334:	MONTH_OF_DATE := 11;
		335..365:	MONTH_OF_DATE := 12;
	END_CASE;
END_IF;


(* old code used in rev 1.0
month := STRING_TO_INT(MID(DATE_TO_STRING(idate),2,8));
*)

(* revision history
hm	1. aug 2006		rev 1.0
	original version	

hm	1. okt 2007		rev 1.1
	replaced old code (string conversion) with mathematics
	the execution time is now multiple times faster.

hm	7. oct. 2008	rev 1.2
	changed name of function from month to MONTH_OF_DATE

*)
END_FUNCTION

(* POU DAY_OF_YEAR, ST *)
FUNCTION DAY_OF_YEAR : INT
VAR_INPUT
	IDATE : DATE;
END_VAR
VAR
END_VAR

(*
version 1.3	7. oct. 2008
programmer 	hugo
tested by	oscat

calculates the day of the year

*)
DAY_OF_YEAR := DWORD_TO_INT((DATE_TO_DWORD(idate) - DATE_TO_DWORD(YEAR_BEGIN(YEAR_OF_DATE(idate))))/86400) + 1;


(* version before rev 1.2
IF step7 THEN
	day_of_year := DWORD_TO_INT(DATE_TO_DWORD(idate)/86400 + 726483 - TRUNC((year(idate)-1)*365.25));
ELSE
	day_of_year := DWORD_TO_INT(DATE_TO_DWORD(idate)/86400 + 719178 - TRUNC((year(idate)-1)*365.25));
END_IF;
*)


(* revivision history
hm	4. aug. 2007		rev 1.0
	original version

hm	1. oct. 2007		rev 1.1
	added compatibility to STEP7

hm	4. jan. 2008		rev 1.2
	changed code for better performance

hm	7. oct. 2008		rev 1.3
	changed name of function year to year_of_date
*)
END_FUNCTION

(* POU YEAR_BEGIN, ST *)
FUNCTION YEAR_BEGIN : DATE
VAR_INPUT
	y : INT;
END_VAR
VAR
END_VAR

(*
version 1.2	7. Apr. 2008
programmer 	hugo
tested by	tobias

returs the date of january 1st for the given year  
the function works for dates from 1970 - 2099 

*)
YEAR_BEGIN := DWORD_TO_DATE(SHR(INT_TO_DWORD(y) * 1461 - 2878169,2)*86400);



(* revision history
hm	19. dec 2007	rev 1.0
	original version

hm	4. jan 2008		rev 1.1
	formula for step7 was incorrect during leap years

hm	7. apr. 2008	rev 1.2
	deleted unused step7 code
*)
END_FUNCTION

(* POU LEAP_OF_DATE, ST *)
FUNCTION LEAP_OF_DATE : BOOL
VAR_INPUT
	idate : DATE;
END_VAR
VAR
END_VAR

(*
version 1.2	8 jan 2008
programmer 	hugo
tested by		tobias

leap_year is true if the tested year is a leap year  

*)
leap_of_Date := SHL(DWORD_TO_INT((DATE_TO_DWORD(idate)+43200) / 31557600)+2,14) = 0;


(* change history

2.10.2006		rev 1.1
the function now calls leap_year to accomodate further accuracy.
the function now works for any year from 1970 to 2100

8. jan 2008		rev 1.2
	improved code for better performance
*)
END_FUNCTION

(* POU FLOOR, ST *)
FUNCTION FLOOR : INT
VAR_INPUT
	X : REAL;
END_VAR
VAR
END_VAR


(*
version 1.1	21. mar. 2008
programmer 	hugo
tested by		tobias

This is a rounding function which returns the biggest possible integer which is less or equal to X.
floor(3.14) = 3
floor(-3.14) = -4

*)
FLOOR := REAL_TO_INT(X);
IF FLOOR > X THEN
	FLOOR := FLOOR - 1;
END_IF;

(* revision history
hm		7. feb 2007		rev 1.0
	originlal version

hm		21. mar. 2008	rev 1.1
	replaced trunc with real_to_int for compatibility reasons

*)
END_FUNCTION

(* POU DAY_OF_MONTH, ST *)
FUNCTION DAY_OF_MONTH : INT
VAR_INPUT
	IDATE : DATE;
END_VAR
VAR
	leap: INT;
END_VAR

(*
version 2.0	25. oct. 2008
programmer 	hugo
tested by	tobias

returns the day OF month for any DATE

*)
(* calculate the day in the year *)
DAY_OF_MONTH := DAY_OF_YEAR(idate);
(* leap will be set to one for a leap year *)
leap := BOOL_TO_INT(LEAP_OF_DATE(idate));
(* if leap year deduct one from the days of the year *)
DAY_OF_MONTH := DAY_OF_MONTH - leap;
(* search if we are in month december to march ? *)
IF DAY_OF_MONTH > setup.MTH_OFS[9] THEN
	IF DAY_OF_MONTH > setup.MTH_OFS[11] THEN
		IF DAY_OF_MONTH > setup.mth_ofs[12] THEN
			DAY_OF_MONTH := DAY_OF_MONTH - setup.MTH_OFS[12];
		ELSE
			DAY_OF_MONTH := DAY_OF_MONTH - setup.MTH_OFS[11];
		END_IF;
	ELSE
		IF DAY_OF_MONTH > setup.mth_ofs[10] THEN
			DAY_OF_MONTH := DAY_OF_MONTH - setup.MTH_OFS[10];
		ELSE
			DAY_OF_MONTH := DAY_OF_MONTH - setup.MTH_OFS[9];
		END_IF;
	END_IF;
ELSIF DAY_OF_MONTH > setup.MTH_OFS[5] THEN
	IF DAY_OF_MONTH > setup.MTH_OFS[7] THEN
		IF DAY_OF_MONTH > setup.mth_ofs[8] THEN
			DAY_OF_MONTH := DAY_OF_MONTH - setup.MTH_OFS[8];
		ELSE
			DAY_OF_MONTH := DAY_OF_MONTH - setup.MTH_OFS[7];
		END_IF;
	ELSE
		IF DAY_OF_MONTH > setup.mth_ofs[6] THEN
			DAY_OF_MONTH := DAY_OF_MONTH - setup.MTH_OFS[6];
		ELSE
			DAY_OF_MONTH := DAY_OF_MONTH - setup.MTH_OFS[5];
		END_IF;
	END_IF;
ELSIF DAY_OF_MONTH > setup.MTH_OFS[3] THEN
	IF DAY_OF_MONTH > setup.MTH_OFS[4] THEN
		DAY_OF_MONTH := DAY_OF_MONTH - setup.MTH_OFS[4];
	ELSE
		DAY_OF_MONTH := DAY_OF_MONTH - setup.MTH_OFS[3];
	END_IF;
ELSE
	(* since now we must be in february or january we need to add leap again *)
	DAY_OF_MONTH := DAY_OF_MONTH + leap;
	IF DAY_OF_MONTH > setup.MTH_OFS[2] THEN DAY_OF_MONTH := DAY_OF_MONTH - setup.mth_ofs[2]; END_IF;
	(* since nothing was true before, day_of_month must already be good *)
END_IF;



(*
(* this was try number one but a loop is too slow *)
(* calculate the day in the year *)
DAY_OF_MONTH := DAY_OF_YEAR(idate);
(* leap will be set to one for a leap year *)
leap := BOOL_TO_INT(LEAP_OF_DATE(idate));
(* if leap year deduct one from the days of the year *)
DAY_OF_MONTH := DAY_OF_MONTH - leap;
(* search if we are in month december to march ? *)
FOR month := 12 TO 3 BY -1 DO
	IF DAY_OF_MONTH > setup.MTH_OFS[month] THEN
		DAY_OF_MONTH := DAY_OF_MONTH - setup.MTH_OFS[month];
		RETURN;
	END_IF;
END_FOR;
(* since now we must be in february or january we need to add leap again *)
DAY_OF_MONTH := DAY_OF_MONTH + leap;
IF DAY_OF_MONTH > setup.MTH_OFS[2] THEN DAY_OF_MONTH := DAY_OF_MONTH - setup.mth_ofs[2]; END_IF;
(* since nothing was true before, day_of_month must already be good *)
*)





(*
Revision history

hm 22.1.2007		rev 1.1
	deleted unused variable day_in_year and day_in_year_begin

hm	1. okt 2007		rev 1.2
	changed code to use day_of_year and leap_of_date
	added compatibility to STEP7

hm	8. oct 2007		rev 1.3
	deleted unused variable yr

hm	8. jan 2008		rev 1.4
	improved performance

hm	25. oct. 2008	rev 2.0
	new code using setup constants
*)
END_FUNCTION

(* POU SUN_TIME, ST *)
FUNCTION_BLOCK SUN_TIME
VAR_INPUT
	latitude : REAL;				(* latitude of geographical position  *)
	longitude : REAL;				(* longitude of geographical position  *)
	utc : DT;						(*	world time				*)
END_VAR
VAR_OUTPUT
	sun_midday : TOD;			(*	astrological midday in hours when sun stand at south direction	*)
	sun_rise : TOD;				(*	sun rise for current day in local time *)
	sun_set : TOD;				(*	sun set for current day in local time *)
	sun_declination : REAL;		(*	sun declination at midday in degrees	*)
END_VAR
VAR
	T: INT;							(* day in the year   *)
	DK: REAL;						(* sun declination at midday *)
	delta: REAL;					(* delta from midday for sunrise and sunset  *)
	h: REAL;
	B: REAL;
	offset : REAL;
	l15: REAL;
	dat: DATE;
	last_dat: DATE;
END_VAR

(*
version 1.4	17. jan 2008
programmer 	hugo
tested by	tobias

this FUNCTION block calculates the sun rise, sun set, sun offset at midday sun declination for a given date 
for performance reasons the algorithm has been simplified and is accurate within a few minutes only 
the times are calculated in utc and have to be corrected for the given time zone
this correction is not done within sun_time because it would be a problem on days where dst is enabled or disabled


*)
dat := DT_TO_DATE(utc);
IF dat = last_dat THEN RETURN; END_IF;
last_dat := dat;
l15 := longitude * 0.0666666666666;
B := latitude * 0.0174532925199433;
h := -0.0145;
T := day_of_year(dat);
offset := -0.1752 * SIN(0.033430*T + 0.5474) - 0.1340*SIN(0.018234*T - 0.1939);
sun_midday := hour_to_tod(12 + Offset - l15);
DK := 0.40954 * SIN(0.0172 * (T-79.35));
sun_declination := deg(DK);
delta := 12*ACOS((SIN(h) - SIN(B) * SIN(DK)) / (COS(B) * COS(DK))) * 0.318309886;
sun_rise := hour_to_tod(12 - delta - Offset - l15);
sun_set := hour_to_tod(12 + delta - Offset - l15);

(* revision history

rev 1.1	hm	20.1.2007
	deleted unused variables sun_riseR and sun_setR

rev 1.2 hm 17.4.2007
	corrected error while sun:midday would not be corrected for longitude.

rev 1.3	hm	6. jan 2008
	performance improvements

rev	1.4 hm	17. jan 2008
	calculation is now only performed once a day
*)
END_FUNCTION_BLOCK

(* POU HOUR_TO_TOD, ST *)
FUNCTION HOUR_TO_TOD : TOD
VAR_INPUT
	IN : REAL;
END_VAR
VAR
END_VAR

(*
version 1.2	24. feb 2009
programmer 	hugo
tested by		tobias

converts an amount of hours in real to time of day TOD.

*)
HOUR_TO_TOD := DWORD_TO_TOD(REAL_TO_DWORD(IN * 3600000));


(* revision history
hm	4. aug. 2006	rev 1.0
	original version

hm	14. mar. 2008	rev 1.1
	rounded the input after the last digit

hm	24. feb. 2009	rev 1.2
	changed input to IN
*)
END_FUNCTION

(* POU SUN_POS, ST *)
FUNCTION_BLOCK SUN_POS
VAR_INPUT
	latitude : REAL;				(* latitude of geographical position  *)
	longitude : REAL;				(* longitude of geographical position  *)
	utc : DT;						(*	world time				*)
END_VAR
VAR_OUTPUT
	B: REAL;
	HR: REAL;
END_VAR
VAR
	g: REAL;
	a: REAL;
	d: REAL;
	h: REAL;
	t1: REAL;
	last: DWORD;
	n: REAL;
	e: REAL;
	c: REAL;
	tau: REAL;
	sin_d: REAL;
	rlat: REAL;
	sin_lat: REAL;
	cos_lat: REAL;
	cos_tau: REAL;
	cos_d: REAL;
	tx: DWORD;
END_VAR

(*
version 2.0	27. feb. 2009
programmer 	hugo
tested by	oscat

this FUNCTION block calculates the sun position for a given date and time.
the times are calculated in utc and have to be corrected for the given time zone.
B is the angle from north and HR is the highth in degrees.

*)
(* EXIT the routine IF it was executed within 10 seconds which is equal to 0.04 degrees accuracy *)
tx := T_PLC_MS();
IF tx - last < 10000 THEN RETURN; END_IF;
last := tx;

(* n is the julian date and the number of days since 1.1.2000-12:00 midday *)
(* be careful for step7 date startes 1.1.1990 instead of 1.1.1970 *)
(* for step7 this line must change *)
n := DWORD_TO_REAL(DT_TO_DWORD(UTC) - 946728000) * 0.000011574074074074;
g :=MODR(6.240040768 + 0.01720197 * n, math.PI2);
d := MODR(4.89495042 + 0.017202792 * n, math.PI2) + 0.033423055 * SIN(g) + 0.000349066 * SIN(2*g);
e := 0.409087723 - 0.000000006981317008 * n;
cos_d := COS(d);
sin_d := SIN(d);
a := ATAN(COS(e) * sin_d / cos_d);
IF cos_d < 0 THEN a := a + math.PI; END_IF;
c := ASIN(SIN(e) * sin_d);

(* also here we must be very careful utc is from 1.1.1970 for step7 the formula must change *)
tau := RAD(MODR(6.697376 + (n - 0.25) * 0.0657098245037645 + DWORD_TO_REAL(TOD_TO_DWORD(DT_TO_TOD(utc))) * 0.0000002785383333, 24) * 15 + longitude) - a;
rlat := RAD(latitude);
sin_lat := SIN(rlat);
cos_lat := COS(rlat);
cos_tau := COS(tau);
t1 := cos_tau * sin_lat - TAN(c) * cos_lat;
B := ATAN(SIN(tau) / t1);
IF t1< 0 THEN B := B + math.PI2; ELSE B := B + math.PI; END_IF;
B := DEG(MODR(b, math.PI2));
h := DEG(ASIN(COS(C) * cos_tau * cos_lat +SIN(c) * sin_lat));
hr := MODR(h + REFRACTION(h),360);
IF hr >= 180 THEN hr := hr - 360; END_IF;


(* revision history
hm	1. feb 2007	rev 1.0
	original version

hm	6. jan 2008	rev 1.1
	performance improvements

hm	18. jan 2008	rev 1.2
	further performance improvements
	only calculate once every 10 seconds

hm	16. mar. 2008	rev 1.3
	added type conversion to avoid warnings under codesys 3.0

hm	30. jun. 2008	rev 1.4
	added type conversions to avoid warnings under codesys 3.0

hm	18. oct. 2008	rev 1.5
	using math constants

hm	17. dec. 2008	rev 1.6
	angles below horizon are displayed in negative degrees

hm	27. feb. 2009	rev 2.0
	new code with better accuracy

*)
END_FUNCTION_BLOCK

(* POU REFRACTION, ST *)
FUNCTION REFRACTION : REAL
VAR_INPUT
	ELEV : REAL;
END_VAR
VAR
	tmp: REAL;
END_VAR


(*
version 1.0	14. jul. 2008
programmer 	hugo
tested by	oscat

REFRACTION calculates the atmospheric refraction in degrees.
the input angle goes from 0 at the hirizon to 90 at midday.

*)
tmp := 0.017453293 * (90.0 - ELEV);
REFRACTION := -0.017 / TAN(tmp + 10.3 / (tmp + 5.11)) - 8.104417E-003;


(* revision histroy
hm	14. jul. 2008	rev 1.0
	original release


*)	
END_FUNCTION

(* POU UTC_TO_LTIME, ST *)
FUNCTION UTC_TO_LTIME : DT
VAR_INPUT
	UTC : DT;
	DST_ENABLE : BOOL;
	TIME_ZONE_OFFSET : INT;
END_VAR
VAR
	tmp: INT;
END_VAR

(*

version 1.9	27. feb. 2009
programmer 	oscat
tested by		oscat

ltime is a real time clock that uses the system rtc as utc time and calculates and given time zone.
the utc time is supplied on the input UTC.
according to the input variable time_zone_offset when the input dst_enable is true,
the dst on and off times are calculated by a formula for any given year and the time is advanced and reset by one hour
at 02:00 and 03:00 for the last sunday of march and last sunday of october.
the code is high performance and the rtc counts every second.
if more then one time zone is needed by the systen the clock can be started many times by placing more then one function block.

 
*)
tmp := TIME_ZONE_OFFSET * 60 + BOOL_TO_INT(DST_ENABLE AND DST(UTC)) * 3600;
IF tmp < 0 THEN
	tmp := ABS(tmp);
	UTC_TO_LTIME := DWORD_TO_DT(DT_TO_DWORD(UTC) -  INT_TO_DWORD(tmp));
ELSE
	UTC_TO_LTIME := DWORD_TO_DT(DT_TO_DWORD(UTC) +  INT_TO_DWORD(tmp));
END_IF;


(* revision history

hm 2.10.2006	rev 1.1
	corrected an error where dst would be delayed by 0.1second

hm 17.1.2007	rev 1.2
	added utc input instead of internal sysrtcgettime because this would only work on wago.
	dst_enable would not be checked before dst would be enabled.

hm 18.3.2007	rev 1.3
	changed code, dst would not work during first cycle.

hm 24.10.2007	rev 1.4
	changed code because the execution every 100ms can cause major problems if the supplied time was not correct at start.
	use of new dst function

hm 12. nov 2007	rev 1.5
		changed Type of time_zone_offset from time to int to allow for time zones with negative offset

hm	8 dec 2007		rev 1.6
	corrected a problem with time_zone_offset

hm	14. oct. 2008	rev 1.7
	renamed module from LTIME to UTC_TO_LTIME
	changed function weekday to day_of_week
	optimized code for better performance

hm	20. oct. 2008	rev 1.8
	changes type of input TIME_ZONE_OFFSET from real to int, now is in +/-minutes
	deleted outputs DST_ON and WDAY
	converted to function

hm	27. feb. 2009	rev 1.9
	added type conversions to avoid warnings under codesys 3.0

*)
END_FUNCTION

(* POU DST, ST *)
FUNCTION DST : BOOL
VAR_INPUT
	UTC : DT;
END_VAR
VAR
	yr : INT;
	yr4 : DWORD;
	ltc: DWORD;
	idate : DWORD;
END_VAR

(*
version 1.4	7. oct. 2008
programmer 	hugo
tested by	oscat

this functions returns TRUE IF dst TIME is active 
the FUNCTION calculates automatically for any year betweek 1970 AND 2099 
wheather daylight savings is on OR off 
the summertime calculation is done according to european standards.
dst will become TRUE AT 01:00 utc in the morning FOR the respective days 
AND it will become FALSE after daylight savings TIME is switched back end OF october at 01:00 utc

*)
yr := YEAR_OF_DATE(DT_TO_DATE(UTC));
ltc := DT_TO_DWORD(UTC);
idate := DT_TO_DWORD(set_DT(yr,3,31,1,0,0));
yr4 := SHR(5*INT_TO_DWORD(yr),2);
DST := (idate - ((yr4+4) MOD 7)*86400 <= ltc) AND (idate + (214 - (yr4+1) MOD 7)*86400 > ltc);


(*
Equation used TO calculate the beginning OF European Summer TIME:
Sunday (31 - (5*y/4 + 4) mod 7) March at 01.00 UTC
(valid through 2099, courtesy of Robert H. van Gent, EC).

European Summer Time ends (clocks go back) at 01.00 UTC on

    * 29 October 2006
    * 28 October 2007
    * 26 October 2008

Equation used to calculate the end of European Summer Time:
Sunday (31 - (5*y/4 + 1) mod 7) October at 01.00 UTC
(validity AND credits as above).

*)



(* revision history
hm	4. aug 2006	rev 1.0
	original version

hm	24. okt 2007	rev 1.1
	deleted time_zone_offset input because dst is generally at 01:00 utc and not mesz
	uk starts 01:00 utc and also greece

hm	1. dec 2007	rev 1.2
	changed code to improve performance

hm	16. mar. 2008	rev 1.3
	added type conversion to avoid warnings under codesys 3.0
	code improvement for better performance

hm	7. oct. 2008	rev 1.4
	changed name of function year to year_of_date
*)
END_FUNCTION

(* POU SET_DT, ST *)
FUNCTION SET_DT : DT
VAR_INPUT
	year : INT;
	month : INT;
	day : INT;
	hour : INT;
	minute : INT;
	second : INT;
END_VAR
VAR
END_VAR

(*
version 1.5	16 mar 2008
programmer 	hugo
tested by	tobias


creates a date output from year, month and day of month
year must be in the form of 4 digits ie 2006 or 1977.
*)
SET_DT := DWORD_TO_DT(DATE_TO_DWORD(SET_DATE(YEAR, MONTH, day)) + INT_TO_DWORD(SECOND) + INT_TO_DWORD(MINUTE) * 60 + INT_TO_DWORD(HOUR) * 3600);


(* revision history
hm	4. aug. 2006		rev 1.0
	original version

hm		19 sep. 2007	rev 1.1
	use function leap_year to calculate leap year, more exceptions are handled

hm		1. okt 2007		rev 1.2
	added step7 compatibility
	call function set_date

hm		8. oct 2007		rev 1.3
	deleted unused variables count and leap

hm		1. 11 2007		rev 1.4
	converted hour type integer to dword in calculation to avoid overrun on möller ecp4

hm		16. mar 2008	rev 1.5
	added type conversions to avoid warnings under codesys 3.0
*)
END_FUNCTION

(* POU HOUR, ST *)
FUNCTION HOUR : INT
VAR_INPUT
	itod : TOD;
END_VAR
VAR
END_VAR

(*
version 1.1	2 okt 2006
programmer 	hugo
tested by	tobias

extracts the hour of a Time_of_day 
*)
hour := DWORD_TO_INT(TOD_TO_DWORD(itod)/3600000);


(* change history
hm 4. aug 2006	rev 1.0
	original version

hm 2.10.2006 	rev 1.1
	changed name of input to itod

*)
END_FUNCTION

(* POU MINUTE, ST *)
FUNCTION MINUTE : INT
VAR_INPUT
	itod : TOD;
END_VAR
VAR
END_VAR

(*
version 1.1	2 oct 2006
programmer 	hugo
tested by	tobias

extracts the minutes out of TOD truncating the seconds 

*)  
MINUTE := DWORD_TO_INT(TOD_TO_DWORD(itod)/60000 - TOD_TO_DWORD(itod)/3600000 * 60);


(* change history

2.10.2006 changes name of input to itod

*)
END_FUNCTION

(* POU SECOND, ST *)
FUNCTION SECOND : REAL
VAR_INPUT
	itod : TOD;
END_VAR
VAR
END_VAR

(*
version 1.1	2 oct 2006
programmer 	hugo
tested by	oscat

returns the seconds and milliseconds as real of TOD   
 
*)
SECOND := DWORD_TO_REAL(TOD_TO_DWORD(itod) - TOD_TO_DWORD(itod)/60000 * 60000) / 1000;



(* change history

hm	2. oct. 2006 rev 1.1 
	changed name of input to itod

*)
END_FUNCTION

(* POU DAY_OF_DATE, ST *)
FUNCTION DAY_OF_DATE : DINT
VAR_INPUT
	idate : DATE;
END_VAR
VAR
END_VAR


(*
	version 1.3	7. apr. 2008
	programmer 	oscat
	tested BY	oscat

DAY_OF_DATE returns the days since 1.1.1970

*)
DAY_OF_DATE := DWORD_TO_DINT(DATE_TO_DWORD(idate) / 86400);


(* revision history
hm		16.9.2007		rev 1.0
	original version

hm		1. okt 2007		rev 1.1
	added step7 compatibility

hm		22. mar. 2008	rev 1.2
	changed output from int to Dint because the total date range is 49710 days

hm		7. apr. 2008	rev 1.3
	deleted unused step7 code

*)
END_FUNCTION

(* POU CALIBRATE, ST *)
FUNCTION_BLOCK CALIBRATE
VAR_INPUT
	X : REAL;
	CO : BOOL;
	CS : BOOL;
END_VAR
VAR_INPUT CONSTANT
	Y_Offset : REAL;
	Y_Scale : REAL;
END_VAR
VAR_OUTPUT
	Y : REAL;
END_VAR
VAR RETAIN
	offset : REAL;
	Scale : REAL := 1;
END_VAR

(*
	version 1.2	22 feb 2007
	programmer 	hugo
	tested BY		hans

Calibrate allows for offset and scale calibration of an analog input.
offset is calibrated to a stored reference Y_offset while CO is true.
after the offset is calibrated, scale can be calibrated to a reference value Y_scale while CS is true.
*)
(* check for calibration *)
IF CO THEN
	Offset := Y_Offset - X;
ELSIF CS THEN
	scale := Y_scale / (X+Offset);
END_IF;
(* calculate output *)
Y := (X + Offset) * Scale;


(* revision history
hm 22.2.2007		rev 1.2
	changed VAR RETAIN PERSISTENT to VAR RETAIN for better compatibility
	wago lon contollers do not support persisitent

*)
END_FUNCTION_BLOCK

(* POU SCALE, ST *)
FUNCTION SCALE : REAL
VAR_INPUT
	X : REAL;
	K : REAL;
	O : REAL;
	MX : REAL;
	MN : REAL;
END_VAR
VAR
END_VAR

(*
version 1.0	16. may. 2008
programmer 	hugo
tested by		tobias

Scale is used to translate an input x to output by the formula Y = X*K + O.
at the same time the output is limited to MN and MX.

*)
SCALE := LIMIT(MN, X * K + O, MX);


(* revision history
hm	16. may. 2008		rev 1.0
	original version
*)
END_FUNCTION

(* POU CAPITALIZE, ST *)
FUNCTION CAPITALIZE : STRING(STRING_LENGTH)
VAR_INPUT
	str : STRING(STRING_LENGTH);
END_VAR
VAR
	PT : POINTER TO BYTE;
	pos : INT;
	L : INT;
	first : BOOL := TRUE;
END_VAR

(*
version 1.2	20. jun. 2008
programmer 	hugo
tested by		tobias

capitalize returns str with all first letters after a blank or beginning of the string are converted to uppercase.

*)
PT := ADR(CAPITALIZE);
CAPITALIZE := str;
L := LEN(str);
FOR pos := 1 TO l DO
	IF first THEN pt^ := TO_UPPER(pt^);	END_IF;
	(* remember in first if the next char needs to capitalized *)
	first := pt^= 32;
	PT := pt + 1;
END_FOR;

(* revision histroy
hm		4. mar 2008	rev 1.0
	original release

hm	29. mar. 2008	rev 1.1
	changed STRING to STRING(STRING_LENGTH)

hm	20. jun. 2008	rev 1.2
	improved performance

*)	
END_FUNCTION

(* POU TO_UPPER, ST *)
FUNCTION TO_UPPER : BYTE
VAR_INPUT
	IN : BYTE;
END_VAR
VAR
END_VAR

(*
version 1.3	16. jan. 2009
programmer 	hugo
tested by		oscat

to_upper converts a character from lowercase to uppercase

*)
IF in > 96 AND in < 123 THEN
   TO_UPPER := in AND 16#DF;
ELSIF in > 223 AND in <> 247 AND in <> 255 AND setup.EXTENDED_ASCII THEN
   TO_UPPER := in AND 16#DF;
ELSE
   TO_UPPER := in;
END_IF;




(* revision history
hm	6. mar. 2008	rev 1.0
	original version

hm	19. oct. 2008	rev 1.1
	changed setup constants

ks	25. oct. 2008	rev 1.2
	optimized code

hm 16. jan 2009	rev 1.3
	corrected an error in module

*)
END_FUNCTION

(* POU CARG, ST *)
FUNCTION CARG : REAL
VAR_INPUT
	X : complex;
END_VAR
VAR
END_VAR

(*
version 1.1	20. apr. 2008
programmer 	hugo
tested by	oscat

this function calculates the phase angle (argument) of a complex number

*)
CARG := ATAN2(X.im, X.re);



(* revision history
hm	21. feb. 2008	rev 1.0
	original version

hm	20. apr. 2008	rev 1.1
	use ATAN2 instead of ATAN
*)
END_FUNCTION

(* POU CASIN, ST *)
FUNCTION CASIN : complex
VAR_INPUT
	X : complex;
END_VAR
VAR
	Y : complex;
END_VAR

(*
version 1.0	21 feb 2008
programmer 	hugo
tested by	oscat

this function calculates the arcus sinus function of a complex number

*)
y.re := -x.im;
y.im := x.re;
y := CASINH(y);
CASIN.re := y.im;
CASIN.im := -y.re;



(* revision history
hm	21. feb 2008	rev 1.0
	original version


*)
END_FUNCTION

(* POU CASINH, ST *)
FUNCTION CASINH : complex
VAR_INPUT
	X : complex;
END_VAR
VAR
	Y : complex;
END_VAR

(*
version 1.0	21 feb 2008
programmer 	hugo
tested by	oscat

this function calculates the hyperbolic arcus sinus function of a complex number

*)
y.re := (X.re - X.im)*(X.re + X.im) + 1.0;
y.im := 2.0 * X.re * X.im;
y    := CSQRT(y);
y.re := y.re + x.re;
y.im := y.im + x.im;
CASINH  := CLOG(y);



(* revision history
hm	21. feb 2008	rev 1.0
	original version


*)
END_FUNCTION

(* POU CATAN, ST *)
FUNCTION CATAN : complex
VAR_INPUT
	X : complex;
END_VAR
VAR
	r2: REAL;
	num, den : REAL;
END_VAR

(*
version 1.0	21 feb 2008
programmer 	hugo
tested by	oscat

this function calculates the complex arcus tangens

*)
r2 := x.re * x.re;
den := 1.0 - r2 - x.im * x.im;
CATAN.re := 0.5 * ATAN(2.0 * x.re / den);
num := x.im + 1.0;
num := r2 + num * num;
den := x.im - 1.0;
den := r2 + den * den;
CATAN.im := 0.25 * (LN(num)-LN(den));

(* revision history
hm	21. feb 2008	rev 1.0
	original version


*)
END_FUNCTION

(* POU CATANH, ST *)
FUNCTION CATANH : complex
VAR_INPUT
	X : complex;
END_VAR
VAR
	i2: REAL;
	num, den : REAL;
END_VAR

(*
version 1.0	21 feb 2008
programmer 	hugo
tested by	oscat

this function calculates the complex arcus hyperbolic tangens

*)
i2 := x.im * x.im;
num := 1.0 + x.re;
num := i2 + num * num;
den := 1.0 - x.re;
den := i2 + den * den;
CATANH.re := 0.25 * (LN(num) - LN(den));
den := 1 - x.re * x.re - i2;
CATANH.im := 0.5 * ATAN(2.0 * x.im / den);

(* revision history
hm	21. feb 2008	rev 1.0
	original version


*)
END_FUNCTION

(* POU CAUCHY, ST *)
FUNCTION CAUCHY : REAL
VAR_INPUT
	X : REAL;
	T : REAL;
	U : REAL;
END_VAR
VAR
	tmp: REAL;
END_VAR


(*
version 1.0	26. oct. 2008
programmer 	hugo
tested by		tobias

this function calculates the Cauchy distribution function

*)
tmp := x - t;
CAUCHY := math.PI_INV * U / (U*U + tmp*tmp);



(* revision hisdtory
hm	26. oct. 2008	rev 1.0
	original version

*)
END_FUNCTION

(* POU CAUCHYCD, ST *)
FUNCTION CAUCHYCD : REAL
VAR_INPUT
	X : REAL;
	T : REAL;
	U : REAL;
END_VAR
VAR
END_VAR


(*
version 1.0	26. oct. 2008
programmer 	hugo
tested by		tobias

this function calculates the Cauchy distribution function

*)
CAUCHYCD := 0.5 + math.PI_INV * ATAN((X - T) / U);



(* revision hisdtory
hm	26. oct. 2008	rev 1.0
	original version

*)
END_FUNCTION

(* POU CCON, ST *)
FUNCTION CCON : complex
VAR_INPUT
	X : complex;
END_VAR
VAR
END_VAR

(*
version 1.0	21 feb 2008
programmer 	hugo
tested by	oscat

this function calcucates the conjugation of a complex number

*)
CCON.re := x.re;
CCON.im := -x.im;


(* revision history
hm	21. feb 2008	rev 1.0
	original version

*)
END_FUNCTION

(* POU CCOS, ST *)
FUNCTION CCOS : complex
VAR_INPUT
	X : complex;
END_VAR
VAR
END_VAR

(*
version 1.0	21 feb 2008
programmer 	hugo
tested by	oscat

this function calculates the cosinus function of a complex number

*)
CCOS := CCOSH(CSET(-X.im, X.re));


(* revision history
hm	21. feb 2008	rev 1.0
	original version

*)
END_FUNCTION

(* POU CCOSH, ST *)
FUNCTION CCOSH : complex
VAR_INPUT
	X : complex;
END_VAR
VAR
END_VAR

(*
version 1.0	21 feb 2008
programmer 	hugo
tested by	oscat

this function calculates the arcus tangens function of a complex number

*)
CCOSH.re := cosH(x.re) * COS(x.im);
CCOSH.im := sinH(x.re) * SIN(x.im);


(* revision history
hm	21. feb 2008	rev 1.0
	original version

*)
END_FUNCTION

(* POU COSH, ST *)
FUNCTION COSH : REAL
VAR_INPUT
	X : REAL;
END_VAR
VAR
	t: REAL;
END_VAR


(*
version 1.2	5. jan 2008
programmer 	hugo
tested by		tobias

this function calculates the cos hyperbolicus

*)
T := EXP(X);
COSH := (1/T + T) * 0.5;

(* revision histroy
hm	12.1.2007	rev 1.0
	original version

hm	1.12.2007	rev 1.1
	changed code to improve performance

hm	5. jan 2008	rev 1.2
	further performance improvement
*)
END_FUNCTION

(* POU SINH, ST *)
FUNCTION SINH : REAL
VAR_INPUT
	X : REAL;
END_VAR
VAR
END_VAR


(*
version 1.3	11. mar 2008
programmer 	hugo
tested by	tobias

this function calculates the sin hyperbolicus

*)
IF ABS(x) < 2E-3 THEN
	SINH := X;
ELSE
	SINH := (EXP(x) - EXP(-x)) * 0.5;
END_IF;


(* revision history
hm	12.1.2007	rev 1.0
	original version

hm	1.12.2007	rev 1.1
	changed code to improve performance

hm	5. jan 2008	rev 1.2
	further performance improvement

hm	11. mar 2008	rev 1.3
	improved accuracy around 0

*)
END_FUNCTION

(* POU CSET, ST *)
FUNCTION CSET : complex
VAR_INPUT
	RE : REAL;
	IM : REAL;
END_VAR
VAR
END_VAR

(*
version 1.0	21 feb 2008
programmer 	hugo
tested by	oscat

this function creates a complex number from two real inputs

*)
CSET.re := RE;
CSET.im := IM;

(* revision history
hm	21. feb 2008	rev 1.0
	original version

*)
END_FUNCTION

(* POU CDIV, ST *)
FUNCTION CDIV : complex
VAR_INPUT
	X, Y : complex;
END_VAR
VAR
	Temp : REAL;
END_VAR

(*
version 1.0	21 feb 2008
programmer 	hugo
tested by	oscat

